KUKA KRL program: MyProgram_051().src

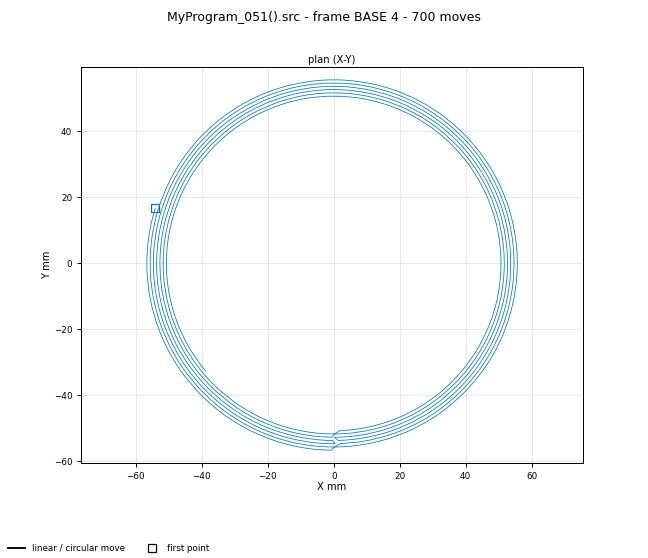
[picture p0: tool path of MyProgram_051().src in frame BASE 4, 700 of 700 moves have a stored position in this frame; points joined in program order, loops and branches not executed]
&ACCESS RVP
&REL 1
&PARAM TEMPLATE = C:\KRC\Roboter\Template\vorgabe
&PARAM EDITMASK = *
DEF MyProgram_051()
; ---- Setting reference (Base) ----
$BASE = BASE_DATA[4]

; --------------------------
; ---- Setting tool (TCP) ----
$TOOL = TOOL_DATA[3]
; --------------------------

$VEL.CP = VEL_APROX_PRINT
Startdeposition()
$VEL.CP = VEL_PRINT
LIN {X -54.1221,Y 16.7008,Z 67,A 157.6929,B 24.8675,C -2.6568,E1 24.846,E2 286.0858} C_DIS
LIN {X -55.301,Y 12.245,Z 67,A 161.7731,B 24.8699,C -2.6326,E1 24.8433,E2 282.0395} C_DIS
LIN {X -55.8838,Y 9.2265,Z 67,A 165.4414,B 24.8699,C -2.6321,E1 24.8415,E2 278.3507} C_DIS
LIN {X -56.3242,Y 5.9752,Z 67,A 168.1233,B 24.872,C -2.6111,E1 24.8406,E2 275.7029} C_DIS
LIN {X -56.6148,Y 1.6943,Z 67,A 172.8319,B 24.8727,C -2.6035,E1 24.8398,E2 270.9843} C_DIS
LIN {X -56.6219,Y -1.4652,Z 67,A 175.993,B 24.8738,C -2.5928,E1 24.8398,E2 267.8296} C_DIS
LIN {X -56.5443,Y -3.2994,Z 67,A 178.54,B 24.8732,C -2.5985,E1 24.8403,E2 265.2537} C_DIS
LIN {X -56.0863,Y -7.9019,Z 67,A -177.3263,B 24.8755,C -2.5749,E1 24.8417,E2 261.1517} C_DIS
LIN {X -55.5998,Y -10.8064,Z 67,A -174.3733,B 24.8765,C -2.5653,E1 24.8431,E2 258.2041} C_DIS
LIN {X -55.076,Y -13.2208,Z 67,A -171.0837,B 24.8759,C -2.5711,E1 24.8453,E2 254.8814} C_DIS
LIN {X -53.9542,Y -17.2366,Z 67,A -167.7374,B 24.8785,C -2.5439,E1 24.8479,E2 251.5808} C_DIS
LIN {X -53.1528,Y -19.5683,Z 67,A -165.0978,B 24.879,C -2.5391,E1 24.8504,E2 248.9377} C_DIS
LIN {X -51.9771,Y -22.5057,Z 67,A -162.0223,B 24.88,C -2.528,E1 24.8537,E2 245.8717} C_DIS
LIN {X -50.9065,Y -24.8344,Z 67,A -159.21,B 24.8804,C -2.5246,E1 24.8571,E2 243.0523} C_DIS
LIN {X -49.5347,Y -27.4672,Z 67,A -156.3958,B 24.8814,C -2.5133,E1 24.8607,E2 240.2501} C_DIS
LIN {X -48.1857,Y -29.7712,Z 67,A -153.4781,B 24.8817,C -2.5101,E1 24.865,E2 237.3252} C_DIS
LIN {X -46.639,Y -32.1398,Z 67,A -150.7212,B 24.8826,C -2.5011,E1 24.8692,E2 234.5758} C_DIS
LIN {X -45.2413,Y -34.0785,Z 67,A -147.4375,B 24.8817,C -2.5105,E1 24.8748,E2 231.2539} C_DIS
LIN {X -41.3308,Y -38.7283,Z 67,A -141.1779,B 24.8828,C -2.499,E1 24.8864,E2 224.9939} C_DIS
LIN {X -39.0762,Y -41.0032,Z 67,A -137.9651,B 24.8834,C -2.4919,E1 24.8929,E2 221.7846} C_DIS
LIN {X -35.9928,Y -43.7344,Z 67,A -134.4049,B 24.8852,C -2.4731,E1 24.9004,E2 218.2555} C_DIS
LIN {X -33.4392,Y -45.7158,Z 67,A -131.3934,B 24.8862,C -2.4628,E1 24.9071,E2 215.2577} C_DIS
LIN {X -31.3897,Y -47.1472,Z 67,A -128.7043,B 24.8862,C -2.4618,E1 24.9133,E2 212.5622} C_DIS
LIN {X -29.065,Y -48.615,Z 67,A -125.9136,B 24.8866,C -2.4579,E1 24.92,E2 209.772} C_DIS
LIN {X -26.584,Y -50.0145,Z 67,A -123.2284,B 24.8873,C -2.4505,E1 24.9265,E2 207.0968} C_DIS
LIN {X -24.2627,Y -51.1812,Z 67,A -120.5751,B 24.8875,C -2.4478,E1 24.9332,E2 204.4429} C_DIS
LIN {X -20.1408,Y -52.9383,Z 67,A -115.6937,B 24.8874,C -2.4499,E1 24.9458,E2 199.5456} C_DIS
LIN {X -16.9667,Y -54.0396,Z 67,A -112.4919,B 24.8879,C -2.4435,E1 24.9543,E2 196.3531} C_DIS
LIN {X -14.3599,Y -54.7903,Z 67,A -109.8261,B 24.8882,C -2.4403,E1 24.9615,E2 193.6907} C_DIS
LIN {X -11.9749,Y -55.3599,Z 67,A -107.3588,B 24.8884,C -2.4389,E1 24.9682,E2 191.2237} C_DIS
LIN {X -9.3697,Y -55.8598,Z 67,A -104.6044,B 24.8884,C -2.4394,E1 24.9758,E2 188.4653} C_DIS
LIN {X -6.5203,Y -56.2637,Z 67,A -101.862,B 24.8887,C -2.4355,E1 24.9833,E2 185.73} C_DIS
LIN {X -4.0645,Y -56.4947,Z 67,A -99.183,B 24.8883,C -2.4391,E1 24.9908,E2 183.0414} C_DIS
LIN {X -0.895,Y -56.6333,Z 67,A -95.9984,B 24.8883,C -2.4391,E1 24.9997,E2 179.8564} C_DIS
LIN {X -0.895,Y -56.6333,Z 67,A -95.9984,B 24.8883,C -2.4391,E1 24.9997,E2 179.8564} C_DIS
Enddeposition()
LIN {X 0.3106,Y -55.6512,Z 67,A -94.8837,B 24.887,C -2.4541,E1 25.0029,E2 178.706} C_DIS
Startdeposition()
$VEL.CP = VEL_PRINT
LIN {X -1.8445,Y -55.6223,Z 67,A -98.806,B 24.89,C -2.4206,E1 24.9918,E2 182.7081} C_DIS
LIN {X -4.7912,Y -55.447,Z 67,A -101.3708,B 24.8892,C -2.4297,E1 24.9847,E2 185.2525} C_DIS
LIN {X -7.4963,Y -55.1465,Z 67,A -104.2719,B 24.8893,C -2.4282,E1 24.9766,E2 188.159} C_DIS
LIN {X -11.1478,Y -54.5248,Z 67,A -108.48,B 24.8899,C -2.4223,E1 24.965,E2 192.3859} C_DIS
LIN {X -13.8894,Y -53.8916,Z 67,A -110.9193,B 24.889,C -2.4323,E1 24.9585,E2 194.8048} C_DIS
LIN {X -16.4128,Y -53.1775,Z 67,A -113.7184,B 24.889,C -2.4323,E1 24.9509,E2 197.6086} C_DIS
LIN {X -18.8336,Y -52.3696,Z 67,A -116.0432,B 24.8883,C -2.4399,E1 24.9448,E2 199.9195} C_DIS
LIN {X -21.0409,Y -51.5219,Z 67,A -118.81,B 24.8886,C -2.4362,E1 24.9376,E2 202.7012} C_DIS
LIN {X -23.8797,Y -50.2697,Z 67,A -121.8951,B 24.8881,C -2.4417,E1 24.9298,E2 205.7808} C_DIS
LIN {X -26.7603,Y -48.7973,Z 67,A -124.7977,B 24.887,C -2.4535,E1 24.9227,E2 208.6632} C_DIS
LIN {X -29.3984,Y -47.2542,Z 67,A -128.3435,B 24.8873,C -2.4509,E1 24.9141,E2 212.226} C_DIS
LIN {X -31.6691,Y -45.7635,Z 67,A -131.1634,B 24.8869,C -2.4549,E1 24.9076,E2 215.0458} C_DIS
LIN {X -34.5559,Y -43.6247,Z 67,A -134.6556,B 24.886,C -2.4649,E1 24.8998,E2 218.5269} C_DIS
LIN {X -36.5148,Y -41.9989,Z 67,A -138.1181,B 24.8868,C -2.4554,E1 24.8924,E2 222.0254} C_DIS
LIN {X -40.0607,Y -38.6311,Z 67,A -142.3125,B 24.8846,C -2.4799,E1 24.8841,E2 226.1788} C_DIS
LIN {X -41.1545,Y -37.4636,Z 67,A -144.6872,B 24.8854,C -2.4713,E1 24.8796,E2 228.5847} C_DIS
LIN {X -44.1926,Y -33.827,Z 67,A -149.3108,B 24.8839,C -2.4868,E1 24.8715,E2 233.1927} C_DIS
LIN {X -45.5071,Y -32.038,Z 67,A -151.4004,B 24.8831,C -2.4956,E1 24.8681,E2 235.2717} C_DIS
LIN {X -47.4442,Y -29.0915,Z 67,A -154.6624,B 24.8817,C -2.5108,E1 24.8632,E2 238.5137} C_DIS
LIN {X -48.5041,Y -27.2875,Z 67,A -157.3262,B 24.8819,C -2.5081,E1 24.8595,E2 241.1977} C_DIS
LIN {X -49.835,Y -24.7729,Z 67,A -160.2896,B 24.8812,C -2.5155,E1 24.8557,E2 244.1595} C_DIS
LIN {X -51.5972,Y -20.856,Z 67,A -164.7992,B 24.8802,C -2.5265,E1 24.8507,E2 248.6677} C_DIS
LIN {X -52.3478,Y -18.8934,Z 67,A -166.8741,B 24.8795,C -2.5341,E1 24.8487,E2 250.7361} C_DIS
LIN {X -53.23,Y -16.2436,Z 67,A -170.2299,B 24.8794,C -2.5349,E1 24.8459,E2 254.1092} C_DIS
LIN {X -54.2859,Y -12.2611,Z 67,A -173.8372,B 24.8772,C -2.5577,E1 24.8434,E2 257.6831} C_DIS
LIN {X -54.8971,Y -9.137,Z 67,A -177.5377,B 24.8769,C -2.561,E1 24.8416,E2 261.3975} C_DIS
LIN {X -55.3786,Y -5.5122,Z 67,A 178.4718,B 24.8761,C -2.5692,E1 24.8403,E2 265.3924} C_DIS
LIN {X -55.6028,Y -2.3569,Z 67,A 175.2683,B 24.875,C -2.5802,E1 24.8398,E2 268.5889} C_DIS
LIN {X -55.6332,Y 1.4878,Z 67,A 171.6315,B 24.8733,C -2.5977,E1 24.8398,E2 272.2058} C_DIS
LIN {X -55.4904,Y 4.2453,Z 67,A 169.0616,B 24.872,C -2.6109,E1 24.8403,E2 274.7594} C_DIS
LIN {X -55.353,Y 5.7673,Z 67,A 167.1882,B 24.872,C -2.6112,E1 24.8408,E2 276.6435} C_DIS
LIN {X -55.0287,Y 8.313,Z 67,A 164.6327,B 24.871,C -2.6208,E1 24.8418,E2 279.1912} C_DIS
LIN {X -54.6417,Y 10.5596,Z 67,A 161.8621,B 24.871,C -2.6216,E1 24.8432,E2 281.9764} C_DIS
LIN {X -53.7999,Y 14.2433,Z 67,A 157.9782,B 24.8698,C -2.6337,E1 24.8458,E2 285.854} C_DIS
LIN {X -53.2007,Y 16.3381,Z 67,A 155.4974,B 24.8694,C -2.6369,E1 24.8479,E2 288.3415} C_DIS
LIN {X -52.3409,Y 18.9123,Z 67,A 152.2747,B 24.8693,C -2.6387,E1 24.8509,E2 291.5781} C_DIS
LIN {X -50.5816,Y 23.2124,Z 67,A 148.3561,B 24.8665,C -2.6664,E1 24.8552,E2 295.4521} C_DIS
LIN {X -49.413,Y 25.6061,Z 67,A 145.5521,B 24.8658,C -2.6734,E1 24.8587,E2 298.2545} C_DIS
LIN {X -48.1498,Y 27.9081,Z 67,A 142.8105,B 24.8651,C -2.6805,E1 24.8625,E2 300.9935} C_DIS
LIN {X -46.6638,Y 30.3274,Z 67,A 139.9688,B 24.8641,C -2.6899,E1 24.8667,E2 303.8273} C_DIS
LIN {X -44.8507,Y 32.9491,Z 67,A 136.9036,B 24.8629,C -2.7022,E1 24.8716,E2 306.8781} C_DIS
LIN {X -43.6109,Y 34.5734,Z 67,A 134.4878,B 24.8629,C -2.7026,E1 24.8758,E2 309.3042} C_DIS
LIN {X -41.8572,Y 36.677,Z 67,A 131.7034,B 24.862,C -2.7103,E1 24.8808,E2 312.083} C_DIS
LIN {X -39.6827,Y 39.0195,Z 67,A 128.1736,B 24.8616,C -2.7143,E1 24.8876,E2 315.6185} C_DIS
LIN {X -37.3353,Y 41.272,Z 67,A 124.9518,B 24.8606,C -2.7241,E1 24.8942,E2 318.8301} C_DIS
LIN {X -35.221,Y 43.0901,Z 67,A 122.1383,B 24.8599,C -2.7313,E1 24.9002,E2 321.6372} C_DIS
LIN {X -33.067,Y 44.7644,Z 67,A 119.0584,B 24.8598,C -2.7325,E1 24.9071,E2 324.7253} C_DIS
LIN {X -29.6626,Y 47.0892,Z 67,A 115.4695,B 24.8578,C -2.7517,E1 24.9153,E2 328.2803} C_DIS
LIN {X -26.8663,Y 48.7393,Z 67,A 111.6008,B 24.8581,C -2.7485,E1 24.9247,E2 332.1681} C_DIS
LIN {X -24.4566,Y 49.9918,Z 67,A 108.8439,B 24.8576,C -2.7536,E1 24.9316,E2 334.9201} C_DIS
LIN {X -21.7856,Y 51.2118,Z 67,A 105.258,B 24.8581,C -2.7483,E1 24.9408,E2 338.5272} C_DIS
LIN {X -18.7901,Y 52.3853,Z 67,A 102.8014,B 24.8561,C -2.7675,E1 24.9471,E2 340.9433} C_DIS
LIN {X -15.8274,Y 53.3546,Z 67,A 98.6582,B 24.8575,C -2.7546,E1 24.9583,E2 345.1243} C_DIS
LIN {X -12.7972,Y 54.1618,Z 67,A 95.4033,B 24.8572,C -2.7571,E1 24.9671,E2 348.3777} C_DIS
LIN {X -7.566,Y 55.1364,Z 67,A 90.5156,B 24.8557,C -2.7717,E1 24.9805,E2 353.2354} C_DIS
LIN {X -4.5272,Y 55.4683,Z 67,A 87.2828,B 24.8557,C -2.7717,E1 24.9894,E2 356.4699} C_DIS
LIN {X -1.7783,Y 55.6243,Z 67,A 84.466,B 24.8556,C -2.7729,E1 24.9973,E2 359.2843} C_DIS
LIN {X 1.3657,Y 55.637,Z 67,A 81.6491,B 24.8547,C -2.7813,E1 25.0051,E2 362.0811} C_DIS
LIN {X 3.1678,Y 55.5625,Z 67,A 79.4313,B 24.8554,C -2.7746,E1 25.0113,E2 364.3141} C_DIS
LIN {X 5.966,Y 55.3322,Z 67,A 76.2287,B 24.856,C -2.7684,E1 25.0203,E2 367.5295} C_DIS
LIN {X 10.5629,Y 54.6411,Z 67,A 71.7775,B 24.8555,C -2.7733,E1 25.0325,E2 371.9646} C_DIS
LIN {X 13.0854,Y 54.0926,Z 67,A 68.9473,B 24.856,C -2.7685,E1 25.0402,E2 374.8021} C_DIS
LIN {X 15.7507,Y 53.3774,Z 67,A 66.5106,B 24.8554,C -2.7746,E1 25.0467,E2 377.2205} C_DIS
LIN {X 18.0833,Y 52.6324,Z 67,A 63.5248,B 24.8566,C -2.7634,E1 25.0547,E2 380.2271} C_DIS
LIN {X 20.7445,Y 51.6425,Z 67,A 60.8487,B 24.8564,C -2.7655,E1 25.0616,E2 382.8924} C_DIS
LIN {X 23.7433,Y 50.3345,Z 67,A 57.4715,B 24.8568,C -2.7615,E1 25.0702,E2 386.2705} C_DIS
LIN {X 26.1701,Y 49.1164,Z 67,A 54.7715,B 24.8569,C -2.7599,E1 25.0769,E2 388.9668} C_DIS
LIN {X 28.4356,Y 47.8399,Z 67,A 52.0436,B 24.8574,C -2.7551,E1 25.0835,E2 391.6979} C_DIS
LIN {X 30.7794,Y 46.3668,Z 67,A 49.258,B 24.8577,C -2.752,E1 25.09,E2 394.4817} C_DIS
LIN {X 32.7053,Y 45.0292,Z 67,A 46.9243,B 24.858,C -2.7497,E1 25.0953,E2 396.8128} C_DIS
LIN {X 35.9425,Y 42.4899,Z 67,A 42.7233,B 24.8587,C -2.7427,E1 25.1045,E2 401.0146} C_DIS
LIN {X 38.4218,Y 40.2624,Z 67,A 39.2402,B 24.8595,C -2.7349,E1 25.1117,E2 404.5023} C_DIS
LIN {X 40.6729,Y 37.9865,Z 67,A 36.2169,B 24.8596,C -2.7336,E1 25.1176,E2 407.5155} C_DIS
LIN {X 43.1485,Y 35.149,Z 67,A 32.5217,B 24.8601,C -2.7288,E1 25.1243,E2 411.2054} C_DIS
LIN {X 44.2479,Y 33.754,Z 67,A 29.9013,B 24.8623,C -2.7075,E1 25.1288,E2 413.8638} C_DIS
LIN {X 46.5073,Y 30.5663,Z 67,A 26.43,B 24.8621,C -2.7094,E1 25.1343,E2 417.3136} C_DIS
LIN {X 47.6256,Y 28.7931,Z 67,A 24.4975,B 24.8622,C -2.7088,E1 25.1371,E2 419.2378} C_DIS
LIN {X 48.5299,Y 27.2412,Z 67,A 22.2207,B 24.8636,C -2.6946,E1 25.1403,E2 421.5363} C_DIS
LIN {X 49.765,Y 24.9142,Z 67,A 19.2963,B 24.8649,C -2.6826,E1 25.1441,E2 424.4735} C_DIS
LIN {X 50.9938,Y 22.2902,Z 67,A 16.8273,B 24.8646,C -2.6856,E1 25.1469,E2 426.9222} C_DIS
LIN {X 52.4735,Y 18.541,Z 67,A 12.9781,B 24.8651,C -2.6803,E1 25.1508,E2 430.7625} C_DIS
LIN {X 53.1743,Y 16.4231,Z 67,A 9.8911,B 24.8675,C -2.6561,E1 25.1535,E2 433.8891} C_DIS
LIN {X 53.8261,Y 14.1443,Z 67,A 7.7022,B 24.8677,C -2.6544,E1 25.155,E2 436.0696} C_DIS
LIN {X 54.454,Y 11.4927,Z 67,A 4.92,B 24.8685,C -2.6464,E1 25.1567,E2 438.8546} C_DIS
LIN {X 55.0641,Y 8.0767,Z 67,A 1.1075,B 24.8701,C -2.6301,E1 25.1585,E2 442.6832} C_DIS
LIN {X 55.4353,Y 4.9183,Z 67,A -1.8284,B 24.8704,C -2.6274,E1 25.1593,E2 445.6081} C_DIS
LIN {X 55.5989,Y 2.4463,Z 67,A -4.3077,B 24.871,C -2.621,E1 25.1597,E2 448.0878} C_DIS
LIN {X 55.6492,Y -0.7025,Z 67,A -7.5822,B 24.8721,C -2.61,E1 25.1597,E2 451.3687} C_DIS
LIN {X 55.5487,Y -3.4141,Z 67,A -10.1765,B 24.8725,C -2.6057,E1 25.1594,E2 453.9579} C_DIS
LIN {X 55.3691,Y -5.6137,Z 67,A -12.6549,B 24.8737,C -2.5939,E1 25.1588,E2 456.4495} C_DIS
LIN {X 54.6207,Y -10.6686,Z 67,A -17.6644,B 24.8747,C -2.583,E1 25.1566,E2 461.4554} C_DIS
LIN {X 53.8338,Y -14.1146,Z 67,A -21.8632,B 24.877,C -2.5592,E1 25.1538,E2 465.6861} C_DIS
LIN {X 52.8671,Y -17.3885,Z 67,A -24.9749,B 24.8772,C -2.5573,E1 25.1512,E2 468.7845} C_DIS
LIN {X 51.5397,Y -20.9972,Z 67,A -28.8243,B 24.8781,C -2.5478,E1 25.1474,E2 472.6351} C_DIS
LIN {X 50.5576,Y -23.2629,Z 67,A -31.647,B 24.8795,C -2.534,E1 25.1441,E2 475.4749} C_DIS
LIN {X 49.3194,Y -25.7846,Z 67,A -34.155,B 24.8795,C -2.534,E1 25.141,E2 477.9695} C_DIS
LIN {X 48.0794,Y -28.0304,Z 67,A -37.0219,B 24.8806,C -2.5216,E1 25.137,E2 480.8511} C_DIS
LIN {X 46.3184,Y -30.8518,Z 67,A -40.2414,B 24.8811,C -2.5166,E1 25.1322,E2 484.0662} C_DIS
LIN {X 45.1277,Y -32.569,Z 67,A -42.7948,B 24.8825,C -2.502,E1 25.128,E2 486.6417} C_DIS
LIN {X 42.5488,Y -35.8734,Z 67,A -46.3701,B 24.882,C -2.5069,E1 25.1218,E2 490.1887} C_DIS
LIN {X 40.8122,Y -37.8374,Z 67,A -49.8027,B 24.8842,C -2.4843,E1 25.1153,E2 493.6596} C_DIS
LIN {X 38.8834,Y -39.8163,Z 67,A -52.617,B 24.8847,C -2.4782,E1 25.1097,E2 496.4765} C_DIS
LIN {X 35.7352,Y -42.6646,Z 67,A -56.1642,B 24.884,C -2.4859,E1 25.1024,E2 499.9911} C_DIS
LIN {X 33.6953,Y -44.2937,Z 67,A -59.657,B 24.8861,C -2.4631,E1 25.0946,E2 503.5252} C_DIS
LIN {X 31.2855,Y -46.0266,Z 67,A -62.2486,B 24.8858,C -2.4668,E1 25.0887,E2 506.0991} C_DIS
LIN {X 29.2788,Y -47.329,Z 67,A -64.7057,B 24.8862,C -2.4623,E1 25.0829,E2 508.5589} C_DIS
LIN {X 27.4558,Y -48.4097,Z 67,A -66.8391,B 24.8865,C -2.4594,E1 25.0777,E2 510.6926} C_DIS
LIN {X 24.5983,Y -49.9216,Z 67,A -70.2743,B 24.8872,C -2.4517,E1 25.0692,E2 514.1366} C_DIS
LIN {X 22.1325,Y -51.0626,Z 67,A -73.1308,B 24.8877,C -2.4463,E1 25.0619,E2 516.9988} C_DIS
LIN {X 19.0744,Y -52.2818,Z 67,A -76.7513,B 24.8885,C -2.4371,E1 25.0524,E2 520.6335} C_DIS
LIN {X 16.1825,Y -53.2489,Z 67,A -79.5818,B 24.8883,C -2.4396,E1 25.0449,E2 523.4526} C_DIS
LIN {X 11.9676,Y -54.3508,Z 67,A -84.3187,B 24.8892,C -2.4302,E1 25.032,E2 528.2049} C_DIS
LIN {X 9.1373,Y -54.8975,Z 67,A -87.3514,B 24.8895,C -2.4267,E1 25.0237,E2 531.2429} C_DIS
LIN {X 5.1568,Y -55.4133,Z 67,A -90.8379,B 24.8885,C -2.4369,E1 25.0141,E2 534.7024} C_DIS
LIN {X 2.997,Y -55.572,Z 67,A -93.4015,B 24.8892,C -2.4294,E1 25.0069,E2 537.2828} C_DIS
LIN {X 0.3106,Y -55.6512,Z 67,A -94.883,B 24.887,C -2.4538,E1 25.0029,E2 538.706} C_DIS
Enddeposition()
LIN {X 0.3106,Y -55.6512,Z 67,A -94.883,B 24.887,C -2.4538,E1 25.0029,E2 538.706} C_DIS
Startdeposition()
$VEL.CP = VEL_PRINT
LIN {X 1.9823,Y -54.63,Z 67,A -92.5802,B 24.8844,C -2.4821,E1 25.0095,E2 536.3366} C_DIS
LIN {X 7.2815,Y -54.1787,Z 67,A -86.6921,B 24.8835,C -2.4915,E1 25.0259,E2 530.4302} C_DIS
LIN {X 11.5086,Y -53.4402,Z 67,A -82.6061,B 24.8839,C -2.487,E1 25.0371,E2 526.3599} C_DIS
LIN {X 15.7752,Y -52.34,Z 67,A -78.3873,B 24.8842,C -2.4837,E1 25.0484,E2 522.1557} C_DIS
LIN {X 18.8016,Y -51.3302,Z 67,A -74.9215,B 24.8836,C -2.4904,E1 25.0575,E2 518.681} C_DIS
LIN {X 21.2357,Y -50.3719,Z 67,A -72.2364,B 24.8833,C -2.4931,E1 25.0645,E2 515.9957} C_DIS
LIN {X 23.9977,Y -49.1171,Z 67,A -69.529,B 24.8838,C -2.4882,E1 25.0713,E2 513.3069} C_DIS
LIN {X 25.9093,Y -48.1355,Z 67,A -66.7457,B 24.8824,C -2.503,E1 25.0782,E2 510.4962} C_DIS
LIN {X 28.0377,Y -46.928,Z 67,A -64.5615,B 24.8827,C -2.4996,E1 25.0834,E2 508.3267} C_DIS
LIN {X 30.5521,Y -45.3306,Z 67,A -61.5262,B 24.8823,C -2.5037,E1 25.0906,E2 505.2917} C_DIS
LIN {X 31.8249,Y -44.4463,Z 67,A -59.4378,B 24.8811,C -2.5169,E1 25.0954,E2 503.1795} C_DIS
LIN {X 34.6629,Y -42.2713,Z 67,A -55.9867,B 24.8809,C -2.5185,E1 25.1029,E2 499.7373} C_DIS
LIN {X 36.6555,Y -40.5549,Z 67,A -53.1679,B 24.8802,C -2.526,E1 25.1088,E2 496.9118} C_DIS
LIN {X 38.4223,Y -38.8845,Z 67,A -50.8245,B 24.8801,C -2.5276,E1 25.1135,E2 494.5744} C_DIS
LIN {X 40.1119,Y -37.1398,Z 67,A -48.0166,B 24.8789,C -2.5395,E1 25.1189,E2 491.7506} C_DIS
LIN {X 41.8499,Y -35.1705,Z 67,A -45.1235,B 24.878,C -2.5496,E1 25.1242,E2 488.8468} C_DIS
LIN {X 44.048,Y -32.3739,Z 67,A -41.951,B 24.8782,C -2.5472,E1 25.1296,E2 485.6949} C_DIS
LIN {X 44.9481,Y -31.1121,Z 67,A -39.6945,B 24.8764,C -2.5655,E1 25.1332,E2 483.4062} C_DIS
LIN {X 46.4624,Y -28.8021,Z 67,A -37.0281,B 24.8761,C -2.5685,E1 25.1372,E2 480.7461} C_DIS
LIN {X 48.002,Y -26.1553,Z 67,A -33.9945,B 24.8756,C -2.5738,E1 25.1413,E2 477.7158} C_DIS
LIN {X 49.9347,Y -22.2444,Z 67,A -29.7776,B 24.8751,C -2.5794,E1 25.1464,E2 473.5085} C_DIS
LIN {X 50.5459,Y -20.8195,Z 67,A -27.6895,B 24.8736,C -2.5945,E1 25.1487,E2 471.396} C_DIS
LIN {X 51.7095,Y -17.7312,Z 67,A -24.4821,B 24.8731,C -2.5994,E1 25.1517,E2 468.195} C_DIS
LIN {X 52.63,Y -14.7776,Z 67,A -20.9799,B 24.8716,C -2.6152,E1 25.1545,E2 464.6754} C_DIS
LIN {X 53.2679,Y -12.2805,Z 67,A -18.498,B 24.8712,C -2.6187,E1 25.1561,E2 462.1997} C_DIS
LIN {X 54.0301,Y -8.3088,Z 67,A -13.4497,B 24.8681,C -2.6502,E1 25.1585,E2 457.1065} C_DIS
LIN {X 54.4502,Y -4.8468,Z 67,A -10.1854,B 24.8678,C -2.6529,E1 25.1594,E2 453.8552} C_DIS
LIN {X 54.6616,Y -0.7001,Z 67,A -6.335,B 24.8676,C -2.6554,E1 25.1598,E2 450.0218} C_DIS
LIN {X 54.6069,Y 2.5302,Z 67,A -2.9419,B 24.8665,C -2.6662,E1 25.1595,E2 446.6234} C_DIS
LIN {X 54.4176,Y 5.2003,Z 67,A -0.0277,B 24.8654,C -2.6773,E1 25.1588,E2 443.7} C_DIS
LIN {X 54.0544,Y 8.1511,Z 67,A 2.991,B 24.8646,C -2.6848,E1 25.1577,E2 440.6815} C_DIS
LIN {X 53.451,Y 11.4591,Z 67,A 6.4254,B 24.8638,C -2.6935,E1 25.1558,E2 437.2464} C_DIS
LIN {X 52.8997,Y 13.7819,Z 67,A 9.332,B 24.8621,C -2.71,E1 25.1538,E2 434.3176} C_DIS
LIN {X 51.7356,Y 17.6565,Z 67,A 12.7943,B 24.8626,C -2.7053,E1 25.1509,E2 430.8861} C_DIS
LIN {X 50.523,Y 20.8755,Z 67,A 16.3678,B 24.8616,C -2.7149,E1 25.1473,E2 427.3097} C_DIS
LIN {X 49.6029,Y 22.9749,Z 67,A 19.7066,B 24.8588,C -2.7421,E1 25.1434,E2 423.9246} C_DIS
LIN {X 47.8274,Y 26.4739,Z 67,A 23.1375,B 24.8592,C -2.7383,E1 25.1389,E2 420.521} C_DIS
LIN {X 46.9068,Y 28.0736,Z 67,A 25.2669,B 24.8582,C -2.7475,E1 25.1359,E2 418.3806} C_DIS
LIN {X 45.2055,Y 30.7369,Z 67,A 28.3637,B 24.8578,C -2.7512,E1 25.1312,E2 415.2906} C_DIS
LIN {X 43.6371,Y 32.9256,Z 67,A 31.2361,B 24.857,C -2.7591,E1 25.1264,E2 412.4133} C_DIS
LIN {X 42.0608,Y 34.9166,Z 67,A 33.8427,B 24.8565,C -2.7641,E1 25.1218,E2 409.807} C_DIS
LIN {X 40.4202,Y 36.8039,Z 67,A 36.5279,B 24.8557,C -2.7712,E1 25.1168,E2 407.1168} C_DIS
LIN {X 38.2385,Y 39.0661,Z 67,A 39.5381,B 24.8557,C -2.7722,E1 25.1109,E2 404.1172} C_DIS
LIN {X 36.3351,Y 40.8417,Z 67,A 42.4814,B 24.8546,C -2.7821,E1 25.1048,E2 401.1623} C_DIS
LIN {X 34.3582,Y 42.5183,Z 67,A 45.1302,B 24.8542,C -2.7857,E1 25.0991,E2 398.5151} C_DIS
LIN {X 32.3895,Y 44.0365,Z 67,A 47.5643,B 24.8542,C -2.7866,E1 25.0937,E2 396.0875} C_DIS
LIN {X 29.4791,Y 46.0355,Z 67,A 51.5502,B 24.8529,C -2.7984,E1 25.0844,E2 392.0872} C_DIS
LIN {X 26.8906,Y 47.5947,Z 67,A 54.6311,B 24.8526,C -2.8011,E1 25.077,E2 389.0092} C_DIS
LIN {X 24.5763,Y 48.8303,Z 67,A 57.0754,B 24.8529,C -2.7984,E1 25.071,E2 386.578} C_DIS
LIN {X 21.5913,Y 50.2213,Z 67,A 61.075,B 24.8513,C -2.8133,E1 25.0607,E2 382.5531} C_DIS
LIN {X 19.1158,Y 51.2146,Z 67,A 63.6987,B 24.8514,C -2.8124,E1 25.0539,E2 379.9371} C_DIS
LIN {X 16.4547,Y 52.1306,Z 67,A 66.939,B 24.8506,C -2.8205,E1 25.0453,E2 376.6837} C_DIS
LIN {X 12.0362,Y 53.3243,Z 67,A 71.2728,B 24.8512,C -2.8142,E1 25.0336,E2 372.3714} C_DIS
LIN {X 8.8669,Y 53.9415,Z 67,A 74.9893,B 24.8504,C -2.8219,E1 25.0233,E2 368.6407} C_DIS
LIN {X 6.2275,Y 54.3095,Z 67,A 78.5894,B 24.8487,C -2.8379,E1 25.0133,E2 365.0051} C_DIS
LIN {X 2.6694,Y 54.6009,Z 67,A 81.0955,B 24.8512,C -2.8143,E1 25.0064,E2 362.5561} C_DIS
LIN {X -1.0424,Y 54.6552,Z 67,A 84.8338,B 24.8516,C -2.8108,E1 24.996,E2 358.8265} C_DIS
LIN {X -2.6547,Y 54.6016,Z 67,A 86.9733,B 24.8508,C -2.8185,E1 24.99,E2 356.6681} C_DIS
LIN {X -5.9581,Y 54.3393,Z 67,A 90.1154,B 24.8516,C -2.8108,E1 24.9813,E2 353.5429} C_DIS
LIN {X -7.9298,Y 54.0872,Z 67,A 92.114,B 24.8519,C -2.8079,E1 24.9758,E2 351.5495} C_DIS
LIN {X -10.3945,Y 53.6679,Z 67,A 95.1561,B 24.8513,C -2.8136,E1 24.9674,E2 348.4907} C_DIS
LIN {X -12.7914,Y 53.1478,Z 67,A 97.2945,B 24.8524,C -2.8035,E1 24.9616,E2 346.3735} C_DIS
LIN {X -15.5324,Y 52.4121,Z 67,A 100.8773,B 24.8515,C -2.8113,E1 24.9519,E2 342.7665} C_DIS
LIN {X -18.5545,Y 51.4203,Z 67,A 103.8709,B 24.8526,C -2.8012,E1 24.9441,E2 339.7912} C_DIS
LIN {X -21.0677,Y 50.4427,Z 67,A 106.8461,B 24.8527,C -2.8,E1 24.9364,E2 336.8123} C_DIS
LIN {X -23.8238,Y 49.201,Z 67,A 109.98,B 24.8533,C -2.7946,E1 24.9285,E2 333.6834} C_DIS
LIN {X -26.3414,Y 47.9011,Z 67,A 112.8954,B 24.8539,C -2.7887,E1 24.9213,E2 330.7739} C_DIS
LIN {X -28.1411,Y 46.8663,Z 67,A 115.472,B 24.8536,C -2.7917,E1 24.9151,E2 328.1822} C_DIS
LIN {X -31.1429,Y 44.9267,Z 67,A 118.7379,B 24.8552,C -2.7764,E1 24.9076,E2 324.942} C_DIS
LIN {X -33.2316,Y 43.4047,Z 67,A 121.5719,B 24.8556,C -2.773,E1 24.9012,E2 322.106} C_DIS
LIN {X -35.3519,Y 41.6959,Z 67,A 124.4553,B 24.8562,C -2.7674,E1 24.895,E2 319.2252} C_DIS
LIN {X -37.2321,Y 40.0267,Z 67,A 127.7188,B 24.8557,C -2.7718,E1 24.8883,E2 315.9378} C_DIS
LIN {X -40.9282,Y 36.2389,Z 67,A 132.6533,B 24.8581,C -2.7482,E1 24.8789,E2 311.0382} C_DIS
LIN {X -42.6144,Y 34.2396,Z 67,A 135.4081,B 24.8588,C -2.7414,E1 24.874,E2 308.2868} C_DIS
LIN {X -43.7615,Y 32.76,Z 67,A 137.5181,B 24.8591,C -2.7387,E1 24.8705,E2 306.1733} C_DIS
LIN {X -45.47,Y 30.3447,Z 67,A 140.255,B 24.8606,C -2.7244,E1 24.8661,E2 303.4569} C_DIS
LIN {X -46.3436,Y 28.9923,Z 67,A 142.3432,B 24.8604,C -2.7262,E1 24.863,E2 301.3538} C_DIS
LIN {X -48.2524,Y 25.6914,Z 67,A 146.2615,B 24.8617,C -2.7136,E1 24.8577,E2 297.4452} C_DIS
LIN {X -49.8166,Y 22.5077,Z 67,A 150.1592,B 24.8625,C -2.7056,E1 24.853,E2 293.5454} C_DIS
LIN {X -50.8394,Y 20.0902,Z 67,A 152.8049,B 24.8635,C -2.6957,E1 24.8503,E2 290.9087} C_DIS
LIN {X -52.4082,Y 15.5455,Z 67,A 157.948,B 24.8649,C -2.6819,E1 24.8458,E2 285.7691} C_DIS
LIN {X -53.1864,Y 12.6333,Z 67,A 161.8085,B 24.8648,C -2.6833,E1 24.8432,E2 281.8828} C_DIS
LIN {X -53.8355,Y 9.4901,Z 67,A 164.8061,B 24.8664,C -2.6669,E1 24.8417,E2 278.9066} C_DIS
LIN {X -54.3819,Y 5.5595,Z 67,A 168.4825,B 24.8685,C -2.6461,E1 24.8404,E2 275.2578} C_DIS
LIN {X -54.5701,Y 3.2166,Z 67,A 170.8645,B 24.8694,C -2.6371,E1 24.84,E2 272.8831} C_DIS
LIN {X -54.6509,Y 1.2776,Z 67,A 173.0569,B 24.8698,C -2.6332,E1 24.8398,E2 270.6869} C_DIS
LIN {X -54.6475,Y -1.4145,Z 67,A 176.144,B 24.8703,C -2.6285,E1 24.8399,E2 267.5924} C_DIS
LIN {X -54.4784,Y -4.5092,Z 67,A 179.3286,B 24.8714,C -2.6174,E1 24.8405,E2 264.4153} C_DIS
LIN {X -54.1418,Y -7.5475,Z 67,A -177.4963,B 24.8724,C -2.607,E1 24.8416,E2 261.246} C_DIS
LIN {X -53.6425,Y -10.5264,Z 67,A -174.5405,B 24.8737,C -2.594,E1 24.8431,E2 258.3038} C_DIS
LIN {X -53.0306,Y -13.2656,Z 67,A -171.4096,B 24.8742,C -2.5881,E1 24.8451,E2 255.1685} C_DIS
LIN {X -52.1921,Y -16.2566,Z 67,A -168.1325,B 24.8751,C -2.5788,E1 24.8477,E2 251.8948} C_DIS
LIN {X -51.4239,Y -18.5448,Z 67,A -165.485,B 24.8757,C -2.5734,E1 24.8501,E2 249.2453} C_DIS
LIN {X -50.5403,Y -20.8328,Z 67,A -162.6153,B 24.8759,C -2.5709,E1 24.8531,E2 246.3654} C_DIS
LIN {X -48.5848,Y -25.0568,Z 67,A -158.1155,B 24.8778,C -2.5513,E1 24.8586,E2 241.8879} C_DIS
LIN {X -46.6738,Y -28.4578,Z 67,A -154.2195,B 24.8791,C -2.5375,E1 24.864,E2 238.0048} C_DIS
LIN {X -45.6755,Y -30.034,Z 67,A -151.8455,B 24.8789,C -2.5394,E1 24.8676,E2 235.6141} C_DIS
LIN {X -44.4694,Y -31.7924,Z 67,A -149.3054,B 24.8789,C -2.5391,E1 24.8717,E2 233.0625} C_DIS
LIN {X -42.0307,Y -34.9529,Z 67,A -145.3826,B 24.8803,C -2.525,E1 24.8785,E2 229.155} C_DIS
LIN {X -40.4663,Y -36.7534,Z 67,A -143.2395,B 24.8814,C -2.5134,E1 24.8825,E2 227.0298} C_DIS
LIN {X -39.3468,Y -37.9488,Z 67,A -141.6009,B 24.8819,C -2.5085,E1 24.8856,E2 225.3959} C_DIS
LIN {X -37.6038,Y -39.6772,Z 67,A -138.3358,B 24.8813,C -2.5151,E1 24.8922,E2 222.1015} C_DIS
LIN {X -34.5911,Y -42.3295,Z 67,A -134.4223,B 24.8825,C -2.5021,E1 24.9005,E2 218.2038} C_DIS
LIN {X -31.7218,Y -44.5198,Z 67,A -130.6227,B 24.8831,C -2.496,E1 24.909,E2 214.4053} C_DIS
LIN {X -29.2783,Y -46.1644,Z 67,A -127.5602,B 24.8836,C -2.4908,E1 24.9162,E2 211.3452} C_DIS
LIN {X -27.1162,Y -47.4659,Z 67,A -124.8403,B 24.8838,C -2.4884,E1 24.9228,E2 208.6227} C_DIS
LIN {X -24.621,Y -48.8075,Z 67,A -121.6663,B 24.8838,C -2.4884,E1 24.9307,E2 205.4402} C_DIS
LIN {X -21.8407,Y -50.1125,Z 67,A -118.6326,B 24.8844,C -2.4816,E1 24.9384,E2 202.4154} C_DIS
LIN {X -19.4462,Y -51.0895,Z 67,A -115.723,B 24.8844,C -2.4827,E1 24.946,E2 199.4969} C_DIS
LIN {X -15.5881,Y -52.3956,Z 67,A -111.676,B 24.885,C -2.4754,E1 24.9567,E2 195.4601} C_DIS
LIN {X -13.728,Y -52.9135,Z 67,A -109.4222,B 24.8847,C -2.4785,E1 24.9628,E2 193.1955} C_DIS
LIN {X -10.3145,Y -53.6833,Z 67,A -106.0533,B 24.8854,C -2.4713,E1 24.972,E2 189.8396} C_DIS
LIN {X -7.1477,Y -54.196,Z 67,A -102.6592,B 24.8854,C -2.4711,E1 24.9814,E2 186.4432} C_DIS
LIN {X -4.4515,Y -54.4837,Z 67,A -98.7542,B 24.8835,C -2.4915,E1 24.9924,E2 182.4878} C_DIS
LIN {X -0.9847,Y -54.6563,Z 67,A -96.4311,B 24.8858,C -2.4664,E1 24.9987,E2 180.224} C_DIS
LIN {X 0.293,Y -54.6599,Z 67,A -94.8409,B 24.8853,C -2.4717,E1 25.0032,E2 178.6214} C_DIS
Enddeposition()
LIN {X 0.293,Y -54.6599,Z 67,A -94.8409,B 24.8853,C -2.4717,E1 25.0032,E2 178.6214} C_DIS
Startdeposition()
$VEL.CP = VEL_PRINT
LIN {X -0.3288,Y -53.6767,Z 67,A -96.6339,B 24.8858,C -2.467,E1 24.9981,E2 180.4255} C_DIS
LIN {X -2.0978,Y -53.6371,Z 67,A -99.4692,B 24.8874,C -2.4493,E1 24.9901,E2 183.3033} C_DIS
LIN {X -4.9711,Y -53.447,Z 67,A -102.3312,B 24.887,C -2.4533,E1 24.9822,E2 186.1572} C_DIS
LIN {X -9.3391,Y -52.8593,Z 67,A -106.7682,B 24.8865,C -2.4593,E1 24.9699,E2 190.5838} C_DIS
LIN {X -13.6544,Y -51.9128,Z 67,A -111.0069,B 24.8855,C -2.4702,E1 24.9585,E2 194.8023} C_DIS
LIN {X -16.917,Y -50.9424,Z 67,A -115.5048,B 24.8866,C -2.4576,E1 24.9464,E2 199.3379} C_DIS
LIN {X -20.0736,Y -49.7826,Z 67,A -118.3652,B 24.8852,C -2.4736,E1 24.939,E2 202.1665} C_DIS
LIN {X -21.9813,Y -48.9706,Z 67,A -120.834,B 24.8854,C -2.4715,E1 24.9327,E2 204.6461} C_DIS
LIN {X -24.1395,Y -47.9446,Z 67,A -123.5175,B 24.8853,C -2.4722,E1 24.9259,E2 207.3349} C_DIS
LIN {X -27.4783,Y -46.1116,Z 67,A -127.2814,B 24.8843,C -2.4829,E1 24.9168,E2 211.0844} C_DIS
LIN {X -29.9159,Y -44.5688,Z 67,A -130.476,B 24.884,C -2.4856,E1 24.9093,E2 214.2827} C_DIS
LIN {X -31.6921,Y -43.3233,Z 67,A -132.5392,B 24.8833,C -2.4937,E1 24.9047,E2 216.334} C_DIS
LIN {X -33.8899,Y -41.6267,Z 67,A -136.4054,B 24.8842,C -2.4841,E1 24.8961,E2 220.2373} C_DIS
LIN {X -37.6099,Y -38.2986,Z 67,A -140.9748,B 24.882,C -2.507,E1 24.8869,E2 224.7708} C_DIS
LIN {X -39.1891,Y -36.6815,Z 67,A -143.4871,B 24.8817,C -2.5105,E1 24.882,E2 227.2856} C_DIS
LIN {X -40.7951,Y -34.8862,Z 67,A -146.4903,B 24.8818,C -2.5093,E1 24.8765,E2 230.3052} C_DIS
LIN {X -43.7578,Y -31.0896,Z 67,A -150.8251,B 24.8794,C -2.5343,E1 24.8692,E2 234.601} C_DIS
LIN {X -45.1887,Y -28.9702,Z 67,A -154.0575,B 24.8795,C -2.5332,E1 24.8642,E2 237.8523} C_DIS
LIN {X -47.2458,Y -25.4784,Z 67,A -158.0348,B 24.8779,C -2.5499,E1 24.8587,E2 241.8102} C_DIS
LIN {X -48.3791,Y -23.2542,Z 67,A -161.1169,B 24.8779,C -2.5507,E1 24.8548,E2 244.907} C_DIS
LIN {X -49.4799,Y -20.8094,Z 67,A -164.0251,B 24.8772,C -2.558,E1 24.8516,E2 247.8138} C_DIS
LIN {X -50.7321,Y -17.5388,Z 67,A -167.7275,B 24.8761,C -2.5693,E1 24.848,E2 251.5102} C_DIS
LIN {X -51.7368,Y -14.301,Z 67,A -171.4596,B 24.8752,C -2.5783,E1 24.845,E2 255.2424} C_DIS
LIN {X -52.4823,Y -11.2664,Z 67,A -174.4086,B 24.8736,C -2.5942,E1 24.8432,E2 258.1706} C_DIS
LIN {X -52.7957,Y -9.6911,Z 67,A -176.2787,B 24.8734,C -2.5971,E1 24.8422,E2 260.0449} C_DIS
LIN {X -53.1135,Y -7.7648,Z 67,A -178.4089,B 24.8728,C -2.6028,E1 24.8413,E2 262.1742} C_DIS
LIN {X -53.3669,Y -5.7637,Z 67,A 179.3422,B 24.8723,C -2.608,E1 24.8405,E2 264.424} C_DIS
LIN {X -53.5779,Y -3.2851,Z 67,A 176.568,B 24.8717,C -2.6145,E1 24.84,E2 267.1994} C_DIS
LIN {X -53.6766,Y -0.4567,Z 67,A 173.4294,B 24.8709,C -2.6222,E1 24.8398,E2 270.3383} C_DIS
LIN {X -53.6335,Y 2.1696,Z 67,A 170.5474,B 24.8701,C -2.6299,E1 24.84,E2 273.2194} C_DIS
LIN {X -53.4108,Y 5.3517,Z 67,A 167.1245,B 24.8691,C -2.6403,E1 24.8408,E2 276.6378} C_DIS
LIN {X -52.9329,Y 8.9109,Z 67,A 163.8109,B 24.8671,C -2.6602,E1 24.8422,E2 279.9238} C_DIS
LIN {X -52.5982,Y 10.7107,Z 67,A 161.0457,B 24.8677,C -2.6541,E1 24.8437,E2 282.7198} C_DIS
LIN {X -51.897,Y 13.7142,Z 67,A 158.3342,B 24.8658,C -2.673,E1 24.8455,E2 285.4019} C_DIS
LIN {X -50.9601,Y 16.8658,Z 67,A 154.1495,B 24.8658,C -2.6737,E1 24.849,E2 289.6091} C_DIS
LIN {X -49.81,Y 20.0081,Z 67,A 150.8861,B 24.8642,C -2.689,E1 24.8523,E2 292.8542} C_DIS
LIN {X -48.6028,Y 22.7825,Z 67,A 147.9969,B 24.8627,C -2.7037,E1 24.8555,E2 295.7241} C_DIS
LIN {X -47.7039,Y 24.6104,Z 67,A 145.9171,B 24.8619,C -2.7114,E1 24.8581,E2 297.7965} C_DIS
LIN {X -46.48,Y 26.8499,Z 67,A 142.356,B 24.8624,C -2.7064,E1 24.8631,E2 301.3883} C_DIS
LIN {X -44.9495,Y 29.341,Z 67,A 139.3797,B 24.8613,C -2.7172,E1 24.8675,E2 304.3539} C_DIS
LIN {X -42.6678,Y 32.5701,Z 67,A 135.5534,B 24.8596,C -2.7345,E1 24.8738,E2 308.1575} C_DIS
LIN {X -41.0563,Y 34.5799,Z 67,A 132.2212,B 24.8598,C -2.7325,E1 24.8798,E2 311.5098} C_DIS
LIN {X -39.0346,Y 36.8457,Z 67,A 129.7375,B 24.8577,C -2.7523,E1 24.8844,E2 313.9573} C_DIS
LIN {X -37.3209,Y 38.5805,Z 67,A 126.5774,B 24.858,C -2.7496,E1 24.8907,E2 317.137} C_DIS
LIN {X -35.6492,Y 40.1307,Z 67,A 124.3675,B 24.8571,C -2.7586,E1 24.8952,E2 319.3343} C_DIS
LIN {X -33.5414,Y 41.9091,Z 67,A 120.9112,B 24.8573,C -2.7568,E1 24.9028,E2 322.808} C_DIS
LIN {X -30.6564,Y 44.0622,Z 67,A 117.082,B 24.8564,C -2.7647,E1 24.9114,E2 326.6316} C_DIS
LIN {X -26.4073,Y 46.7335,Z 67,A 111.3519,B 24.8561,C -2.7682,E1 24.9252,E2 332.3707} C_DIS
LIN {X -21.7872,Y 49.058,Z 67,A 106.7706,B 24.8536,C -2.7921,E1 24.9366,E2 336.9068} C_DIS
LIN {X -19.9547,Y 49.831,Z 67,A 104.2612,B 24.8539,C -2.7886,E1 24.9431,E2 339.4302} C_DIS
LIN {X -16.6994,Y 51.0143,Z 67,A 100.6767,B 24.8533,C -2.7949,E1 24.9526,E2 343.0064} C_DIS
LIN {X -13.7228,Y 51.8942,Z 67,A 97.5351,B 24.8526,C -2.8013,E1 24.961,E2 346.1379} C_DIS
LIN {X -11.293,Y 52.4765,Z 67,A 94.7785,B 24.8526,C -2.8021,E1 24.9685,E2 348.896} C_DIS
LIN {X -8.3469,Y 53.0249,Z 67,A 91.4453,B 24.8526,C -2.8021,E1 24.9777,E2 352.2325} C_DIS
LIN {X -5.8647,Y 53.357,Z 67,A 89.0654,B 24.8518,C -2.8088,E1 24.9842,E2 354.5983} C_DIS
LIN {X -3.6346,Y 53.5545,Z 67,A 86.594,B 24.8518,C -2.8084,E1 24.9911,E2 357.0716} C_DIS
LIN {X -0.7469,Y 53.6728,Z 67,A 83.1136,B 24.8525,C -2.8022,E1 25.0009,E2 360.5671} C_DIS
LIN {X 1.9531,Y 53.643,Z 67,A 80.8937,B 24.8512,C -2.8145,E1 25.007,E2 362.7575} C_DIS
LIN {X 4.7069,Y 53.4708,Z 67,A 77.3929,B 24.8523,C -2.8043,E1 25.0168,E2 366.2809} C_DIS
LIN {X 8.2661,Y 53.0374,Z 67,A 73.3586,B 24.8528,C -2.7996,E1 25.028,E2 370.3228} C_DIS
LIN {X 11.5658,Y 52.4163,Z 67,A 69.5857,B 24.8533,C -2.7945,E1 25.0383,E2 374.1031} C_DIS
LIN {X 16.2545,Y 51.1583,Z 67,A 65.1595,B 24.8522,C -2.8051,E1 25.0501,E2 378.4966} C_DIS
LIN {X 18.3491,Y 50.4441,Z 67,A 63.0358,B 24.8519,C -2.8077,E1 25.0557,E2 380.61} C_DIS
LIN {X 20.3012,Y 49.6906,Z 67,A 60.6877,B 24.8524,C -2.8033,E1 25.0618,E2 382.9632} C_DIS
LIN {X 22.6153,Y 48.681,Z 67,A 57.5027,B 24.8537,C -2.7908,E1 25.07,E2 386.1698} C_DIS
LIN {X 24.8774,Y 47.5651,Z 67,A 55.0318,B 24.8536,C -2.7917,E1 25.0761,E2 388.6318} C_DIS
LIN {X 27.3497,Y 46.1876,Z 67,A 51.9721,B 24.8541,C -2.7868,E1 25.0835,E2 391.6941} C_DIS
LIN {X 29.4752,Y 44.8611,Z 67,A 49.4638,B 24.8542,C -2.7859,E1 25.0894,E2 394.1962} C_DIS
LIN {X 31.6774,Y 43.334,Z 67,A 46.3019,B 24.8553,C -2.7752,E1 25.0966,E2 397.3726} C_DIS
LIN {X 33.8406,Y 41.6666,Z 67,A 43.8982,B 24.8548,C -2.7802,E1 25.1018,E2 399.7554} C_DIS
LIN {X 35.4046,Y 40.3463,Z 67,A 41.5032,B 24.8557,C -2.7718,E1 25.1069,E2 402.1609} C_DIS
LIN {X 37.169,Y 38.7269,Z 67,A 38.9517,B 24.8562,C -2.7668,E1 25.1121,E2 404.7139} C_DIS
LIN {X 38.9269,Y 36.9603,Z 67,A 36.346,B 24.8567,C -2.7623,E1 25.1172,E2 407.3192} C_DIS
LIN {X 40.3343,Y 35.4184,Z 67,A 34.2187,B 24.857,C -2.7594,E1 25.1211,E2 409.4437} C_DIS
LIN {X 41.5365,Y 34.0012,Z 67,A 32.2938,B 24.8573,C -2.7561,E1 25.1246,E2 411.3678} C_DIS
LIN {X 42.9996,Y 32.1301,Z 67,A 29.2851,B 24.859,C -2.7403,E1 25.1297,E2 414.3995} C_DIS
LIN {X 44.727,Y 29.6781,Z 67,A 25.6455,B 24.8607,C -2.7233,E1 25.1354,E2 418.0614} C_DIS
LIN {X 47.0291,Y 25.8779,Z 67,A 21.2325,B 24.8613,C -2.7176,E1 25.1416,E2 422.4649} C_DIS
LIN {X 48.6479,Y 22.6865,Z 67,A 17.4456,B 24.8623,C -2.7078,E1 25.1462,E2 426.2546} C_DIS
LIN {X 49.728,Y 20.2095,Z 67,A 14.5567,B 24.8631,C -2.6996,E1 25.1492,E2 429.1471} C_DIS
LIN {X 50.9536,Y 16.8851,Z 67,A 11.0008,B 24.8638,C -2.6933,E1 25.1525,E2 432.6978} C_DIS
LIN {X 51.9829,Y 13.382,Z 67,A 7.6636,B 24.8638,C -2.6937,E1 25.155,E2 436.015} C_DIS
LIN {X 52.7059,Y 10.1672,Z 67,A 3.5412,B 24.8661,C -2.6701,E1 25.1574,E2 440.1693} C_DIS
LIN {X 53.2817,Y 6.4995,Z 67,A -0.5103,B 24.8675,C -2.656,E1 25.159,E2 444.2303} C_DIS
LIN {X 53.5702,Y 3.4031,Z 67,A -3.8531,B 24.8686,C -2.6451,E1 25.1596,E2 447.579} C_DIS
LIN {X 53.6739,Y -0.6978,Z 67,A -7.3367,B 24.8681,C -2.6505,E1 25.1598,E2 451.0289} C_DIS
LIN {X 53.4993,Y -4.3731,Z 67,A -11.2658,B 24.8693,C -2.6381,E1 25.1592,E2 454.9641} C_DIS
LIN {X 53.3391,Y -6.0202,Z 67,A -13.8216,B 24.8716,C -2.6155,E1 25.1584,E2 457.5581} C_DIS
LIN {X 52.6539,Y -10.4361,Z 67,A -17.8296,B 24.8714,C -2.6169,E1 25.1565,E2 461.5394} C_DIS
LIN {X 51.9265,Y -13.6015,Z 67,A -22.0838,B 24.8741,C -2.5892,E1 25.1537,E2 465.8344} C_DIS
LIN {X 50.827,Y -17.2605,Z 67,A -26.0636,B 24.8751,C -2.5788,E1 25.1503,E2 469.8162} C_DIS
LIN {X 49.5507,Y -20.6415,Z 67,A -29.1059,B 24.8746,C -2.5847,E1 25.1472,E2 472.8279} C_DIS
LIN {X 48.591,Y -22.8087,Z 67,A -32.2608,B 24.8766,C -2.5638,E1 25.1435,E2 476.015} C_DIS
LIN {X 47.4852,Y -25.0289,Z 67,A -34.6156,B 24.8767,C -2.5624,E1 25.1405,E2 478.3607} C_DIS
LIN {X 45.8511,Y -27.9101,Z 67,A -37.7091,B 24.8767,C -2.5618,E1 25.1362,E2 481.4397} C_DIS
LIN {X 44.8598,Y -29.4771,Z 67,A -39.9057,B 24.8778,C -2.5516,E1 25.1328,E2 483.6492} C_DIS
LIN {X 43.6076,Y -31.3001,Z 67,A -42.2895,B 24.8784,C -2.5448,E1 25.129,E2 486.0377} C_DIS
LIN {X 42.0812,Y -33.3237,Z 67,A -45.1532,B 24.8794,C -2.5343,E1 25.1241,E2 488.9125} C_DIS
LIN {X 40.5952,Y -35.1194,Z 67,A -47.3933,B 24.8795,C -2.5332,E1 25.1201,E2 491.1451} C_DIS
LIN {X 39.4469,Y -36.4042,Z 67,A -49.0827,B 24.8797,C -2.5317,E1 25.1169,E2 492.8304} C_DIS
LIN {X 37.7194,Y -38.1908,Z 67,A -52.2467,B 24.8813,C -2.5147,E1 25.1106,E2 496.0212} C_DIS
LIN {X 35.9093,Y -39.8978,Z 67,A -54.4153,B 24.8809,C -2.5187,E1 25.1062,E2 498.1716} C_DIS
LIN {X 34.6079,Y -41.0322,Z 67,A -56.2784,B 24.8813,C -2.5142,E1 25.1023,E2 500.0381} C_DIS
LIN {X 32.7868,Y -42.5008,Z 67,A -59.0546,B 24.8824,C -2.5031,E1 25.0961,E2 502.8302} C_DIS
LIN {X 30.7376,Y -44.0058,Z 67,A -61.5635,B 24.8825,C -2.5018,E1 25.0905,E2 505.3333} C_DIS
LIN {X 28.8881,Y -45.2415,Z 67,A -64.0411,B 24.8831,C -2.4952,E1 25.0847,E2 507.8185} C_DIS
LIN {X 27.3043,Y -46.2144,Z 67,A -66.2932,B 24.884,C -2.4862,E1 25.0792,E2 510.085} C_DIS
LIN {X 23.9282,Y -48.0494,Z 67,A -70.1343,B 24.8841,C -2.4846,E1 25.0697,E2 513.9191} C_DIS
LIN {X 20.0297,Y -49.8012,Z 67,A -74.3398,B 24.8841,C -2.485,E1 25.059,E2 518.1136} C_DIS
LIN {X 18.6685,Y -50.3273,Z 67,A -76.1383,B 24.8847,C -2.4781,E1 25.0543,E2 519.9244} C_DIS
LIN {X 16.5123,Y -51.0748,Z 67,A -78.3695,B 24.8847,C -2.4792,E1 25.0484,E2 522.1487} C_DIS
LIN {X 15.048,Y -51.5253,Z 67,A -80.8096,B 24.8863,C -2.4617,E1 25.0418,E2 524.6261} C_DIS
LIN {X 10.389,Y -52.6632,Z 67,A -85.2034,B 24.8854,C -2.471,E1 25.0299,E2 528.992} C_DIS
LIN {X 7.3688,Y -53.1698,Z 67,A -89.0394,B 24.8866,C -2.4578,E1 25.0192,E2 532.8555} C_DIS
LIN {X 4.0368,Y -53.5262,Z 67,A -92.0023,B 24.8857,C -2.4676,E1 25.011,E2 535.7935} C_DIS
LIN {X 1.3822,Y -53.6603,Z 67,A -95.2767,B 24.8866,C -2.4584,E1 25.0018,E2 539.0888} C_DIS
LIN {X 1.3822,Y -53.6603,Z 67,A -95.2767,B 24.8866,C -2.4584,E1 25.0018,E2 539.0888} C_DIS
Enddeposition()
LIN {X 0.2815,Y -52.6861,Z 67,A -95.777,B 24.8838,C -2.4879,E1 25.0006,E2 539.5188} C_DIS
Startdeposition()
$VEL.CP = VEL_PRINT
LIN {X 2.1617,Y -52.6459,Z 67,A -93.1189,B 24.8827,C -2.4999,E1 25.0081,E2 536.8328} C_DIS
LIN {X 3.8226,Y -52.552,Z 67,A -91.0535,B 24.8822,C -2.5055,E1 25.0139,E2 534.755} C_DIS
LIN {X 6.4309,Y -52.2966,Z 67,A -88.3019,B 24.8822,C -2.5053,E1 25.0216,E2 532.0058} C_DIS
LIN {X 8.7268,Y -51.9625,Z 67,A -85.9125,B 24.8822,C -2.5045,E1 25.0281,E2 529.6205} C_DIS
LIN {X 10.5866,Y -51.6157,Z 67,A -83.3116,B 24.8811,C -2.5168,E1 25.0353,E2 526.9936} C_DIS
LIN {X 14.3181,Y -50.7075,Z 67,A -79.5156,B 24.8814,C -2.5136,E1 25.0456,E2 523.2112} C_DIS
LIN {X 16.7314,Y -49.9633,Z 67,A -76.6673,B 24.8809,C -2.5189,E1 25.0531,E2 520.3557} C_DIS
LIN {X 19.5615,Y -48.9255,Z 67,A -73.5808,B 24.8809,C -2.5194,E1 25.0612,E2 517.2745} C_DIS
LIN {X 23.1282,Y -47.3438,Z 67,A -69.4871,B 24.8805,C -2.5228,E1 25.0716,E2 513.183} C_DIS
LIN {X 25.7436,Y -45.9731,Z 67,A -66.182,B 24.8798,C -2.5302,E1 25.0797,E2 509.8699} C_DIS
LIN {X 27.6056,Y -44.8803,Z 67,A -63.9006,B 24.8796,C -2.5331,E1 25.0852,E2 507.5886} C_DIS
LIN {X 29.0833,Y -43.9366,Z 67,A -61.7516,B 24.8787,C -2.5417,E1 25.0902,E2 505.4263} C_DIS
LIN {X 31.425,Y -42.2931,Z 67,A -58.8279,B 24.8785,C -2.5441,E1 25.0969,E2 502.5071} C_DIS
LIN {X 33.2332,Y -40.8879,Z 67,A -55.5642,B 24.8764,C -2.5655,E1 25.104,E2 499.2051} C_DIS
LIN {X 37.0219,Y -37.4918,Z 67,A -50.0533,B 24.8752,C -2.5779,E1 25.1152,E2 493.6875} C_DIS
LIN {X 40.4511,Y -33.7636,Z 67,A -45.3523,B 24.8756,C -2.5746,E1 25.1239,E2 489.0152} C_DIS
LIN {X 41.8743,Y -31.981,Z 67,A -42.7679,B 24.8747,C -2.5834,E1 25.1284,E2 486.4224} C_DIS
LIN {X 43.5424,Y -29.6705,Z 67,A -39.9203,B 24.8744,C -2.5864,E1 25.1329,E2 483.5815} C_DIS
LIN {X 44.5006,Y -28.2138,Z 67,A -37.3696,B 24.8725,C -2.6056,E1 25.1368,E2 480.9983} C_DIS
LIN {X 46.2865,Y -25.1758,Z 67,A -34.2345,B 24.8729,C -2.6016,E1 25.1411,E2 477.8888} C_DIS
LIN {X 47.538,Y -22.7247,Z 67,A -30.7994,B 24.8711,C -2.6198,E1 25.1454,E2 474.429} C_DIS
LIN {X 48.6238,Y -20.2983,Z 67,A -28.0163,B 24.8705,C -2.6261,E1 25.1484,E2 471.6463} C_DIS
LIN {X 49.7079,Y -17.4752,Z 67,A -24.9357,B 24.87,C -2.6316,E1 25.1514,E2 468.5699} C_DIS
LIN {X 50.4638,Y -15.1548,Z 67,A -21.966,B 24.8685,C -2.6466,E1 25.1539,E2 465.5816} C_DIS
LIN {X 51.4418,Y -11.4028,Z 67,A -18.2923,B 24.8683,C -2.648,E1 25.1563,E2 461.9259} C_DIS
LIN {X 51.7926,Y -9.688,Z 67,A -16.184,B 24.8673,C -2.6584,E1 25.1574,E2 459.8053} C_DIS
LIN {X 52.204,Y -7.14,Z 67,A -13.5,B 24.8667,C -2.6646,E1 25.1585,E2 457.1225} C_DIS
LIN {X 52.4718,Y -4.7927,Z 67,A -11.1565,B 24.8664,C -2.6678,E1 25.1592,E2 454.7852} C_DIS
LIN {X 52.5831,Y -3.349,Z 67,A -9.2095,B 24.865,C -2.6808,E1 25.1596,E2 452.819} C_DIS
LIN {X 52.6887,Y -0.4997,Z 67,A -5.9367,B 24.8637,C -2.6943,E1 25.1598,E2 449.5338} C_DIS
LIN {X 52.5692,Y 3.5693,Z 67,A -2.0352,B 24.8634,C -2.6969,E1 25.1593,E2 445.6495} C_DIS
LIN {X 52.3267,Y 6.1786,Z 67,A 1.3756,B 24.8613,C -2.7178,E1 25.1583,E2 442.2093} C_DIS
LIN {X 51.7063,Y 10.1364,Z 67,A 5.8393,B 24.8597,C -2.7335,E1 25.1561,E2 437.7347} C_DIS
LIN {X 50.9167,Y 13.5566,Z 67,A 9.1849,B 24.8595,C -2.7348,E1 25.1539,E2 434.4053} C_DIS
LIN {X 50.1673,Y 16.1094,Z 67,A 11.8152,B 24.8592,C -2.7377,E1 25.1517,E2 431.783} C_DIS
LIN {X 49.5375,Y 17.9528,Z 67,A 14.4336,B 24.8575,C -2.7545,E1 25.1492,E2 429.1396} C_DIS
LIN {X 48.1759,Y 21.3374,Z 67,A 17.9499,B 24.8573,C -2.7561,E1 25.1455,E2 425.6388} C_DIS
LIN {X 46.8481,Y 24.1152,Z 67,A 21.9795,B 24.8549,C -2.7797,E1 25.1404,E2 421.575} C_DIS
LIN {X 44.9922,Y 27.4219,Z 67,A 26.2286,B 24.8535,C -2.793,E1 25.1343,E2 417.316} C_DIS
LIN {X 43.1055,Y 30.3027,Z 67,A 29.3644,B 24.8538,C -2.7895,E1 25.1294,E2 414.204} C_DIS
LIN {X 41.3442,Y 32.6637,Z 67,A 32.2766,B 24.8537,C -2.7911,E1 25.1245,E2 411.3018} C_DIS
LIN {X 39.8694,Y 34.4484,Z 67,A 34.8679,B 24.8529,C -2.7984,E1 25.1198,E2 408.7052} C_DIS
LIN {X 37.8958,Y 36.6083,Z 67,A 38.4501,B 24.8513,C -2.8134,E1 25.1129,E2 405.1029} C_DIS
LIN {X 35.034,Y 39.3561,Z 67,A 42.5111,B 24.8509,C -2.8168,E1 25.1046,E2 401.0503} C_DIS
LIN {X 32.8811,Y 41.1718,Z 67,A 45.3555,B 24.8509,C -2.8181,E1 25.0985,E2 398.2138} C_DIS
LIN {X 30.9653,Y 42.6315,Z 67,A 48.3697,B 24.8495,C -2.8305,E1 25.0916,E2 395.181} C_DIS
LIN {X 28.5598,Y 44.2788,Z 67,A 50.9054,B 24.8503,C -2.8229,E1 25.0858,E2 392.6718} C_DIS
LIN {X 26.4516,Y 45.5699,Z 67,A 54.2823,B 24.8484,C -2.8403,E1 25.0776,E2 389.2639} C_DIS
LIN {X 22.5674,Y 47.6127,Z 67,A 58.9604,B 24.848,C -2.8443,E1 25.066,E2 384.5889} C_DIS
LIN {X 19.5621,Y 48.925,Z 67,A 62.4733,B 24.8477,C -2.8469,E1 25.0569,E2 381.078} C_DIS
LIN {X 16.0542,Y 50.1852,Z 67,A 66.5021,B 24.8474,C -2.8498,E1 25.0463,E2 377.0502} C_DIS
LIN {X 12.5969,Y 51.1623,Z 67,A 69.925,B 24.8481,C -2.8431,E1 25.0371,E2 373.6487} C_DIS
LIN {X 10.6013,Y 51.6127,Z 67,A 72.2207,B 24.8479,C -2.8455,E1 25.0308,E2 371.3503} C_DIS
LIN {X 8.0455,Y 52.0723,Z 67,A 75.2016,B 24.8475,C -2.8493,E1 25.0226,E2 368.3633} C_DIS
LIN {X 5.3147,Y 52.4218,Z 67,A 78.2898,B 24.8472,C -2.8516,E1 25.014,E2 365.2721} C_DIS
LIN {X 3.0163,Y 52.6039,Z 67,A 80.4364,B 24.8479,C -2.8451,E1 25.0081,E2 363.1419} C_DIS
LIN {X 1.1598,Y 52.6778,Z 67,A 82.5268,B 24.8479,C -2.8461,E1 25.0022,E2 361.0494} C_DIS
LIN {X -1.0015,Y 52.6807,Z 67,A 85.0025,B 24.8476,C -2.8478,E1 24.9953,E2 358.5695} C_DIS
LIN {X -3.0666,Y 52.6011,Z 67,A 87.056,B 24.8481,C -2.8436,E1 24.9896,E2 356.5256} C_DIS
LIN {X -5.2938,Y 52.4239,Z 67,A 89.696,B 24.8478,C -2.8462,E1 24.9822,E2 353.8782} C_DIS
LIN {X -8.349,Y 52.0243,Z 67,A 93.5194,B 24.8472,C -2.8523,E1 24.9716,E2 350.037} C_DIS
LIN {X -11.285,Y 51.4675,Z 67,A 96.4108,B 24.8481,C -2.8434,E1 24.9638,E2 347.1635} C_DIS
LIN {X -13.9261,Y 50.8167,Z 67,A 99.2061,B 24.8487,C -2.8377,E1 24.9562,E2 344.3776} C_DIS
LIN {X -15.9805,Y 50.2088,Z 67,A 102.0972,B 24.848,C -2.8447,E1 24.9485,E2 341.4648} C_DIS
LIN {X -20.1832,Y 48.6719,Z 67,A 106.3848,B 24.8497,C -2.8285,E1 24.9374,E2 337.2066} C_DIS
LIN {X -22.5158,Y 47.6376,Z 67,A 109.41,B 24.8497,C -2.8285,E1 24.9297,E2 334.1738} C_DIS
LIN {X -24.7391,Y 46.5218,Z 67,A 111.9856,B 24.8504,C -2.822,E1 24.9233,E2 331.6068} C_DIS
LIN {X -26.6638,Y 45.4455,Z 67,A 114.5647,B 24.8505,C -2.8208,E1 24.9171,E2 329.0229} C_DIS
LIN {X -29.3187,Y 43.7801,Z 67,A 117.7943,B 24.8515,C -2.8116,E1 24.9095,E2 325.8049} C_DIS
LIN {X -31.9484,Y 41.9002,Z 67,A 121.914,B 24.8512,C -2.8142,E1 24.9002,E2 321.6643} C_DIS
LIN {X -34.7391,Y 39.6164,Z 67,A 125.8033,B 24.8522,C -2.8051,E1 24.892,E2 317.7816} C_DIS
LIN {X -37.8967,Y 36.6074,Z 67,A 129.8186,B 24.8546,C -2.7825,E1 24.8841,E2 313.8036} C_DIS
LIN {X -39.6657,Y 34.6828,Z 67,A 133.46,B 24.854,C -2.7879,E1 24.8773,E2 310.1329} C_DIS
LIN {X -41.5682,Y 32.3793,Z 67,A 137.1586,B 24.8541,C -2.7866,E1 24.8709,E2 306.42} C_DIS
LIN {X -43.8733,Y 29.1793,Z 67,A 140.3366,B 24.8572,C -2.7577,E1 24.8659,E2 303.2953} C_DIS
LIN {X -45.2541,Y 26.9883,Z 67,A 143.6002,B 24.8572,C -2.7568,E1 24.8611,E2 300.0173} C_DIS
LIN {X -46.5447,Y 24.6956,Z 67,A 146.0398,B 24.8588,C -2.7422,E1 24.8579,E2 297.5998} C_DIS
LIN {X -47.9936,Y 21.7456,Z 67,A 150.6626,B 24.8582,C -2.7477,E1 24.8524,E2 292.9385} C_DIS
LIN {X -49.2058,Y 18.8436,Z 67,A 153.9644,B 24.8594,C -2.7356,E1 24.8491,E2 289.6471} C_DIS
LIN {X -50.8334,Y 13.865,Z 67,A 158.8086,B 24.8626,C -2.7052,E1 24.8451,E2 284.8477} C_DIS
LIN {X -51.31,Y 11.9816,Z 67,A 161.206,B 24.8628,C -2.703,E1 24.8435,E2 282.4417} C_DIS
LIN {X -51.8621,Y 9.3049,Z 67,A 164.1854,B 24.8637,C -2.6938,E1 24.8419,E2 279.4666} C_DIS
LIN {X -52.2921,Y 6.4658,Z 67,A 167.2798,B 24.8648,C -2.6835,E1 24.8408,E2 276.3783} C_DIS
LIN {X -52.5864,Y 3.303,Z 67,A 171.2407,B 24.8651,C -2.6803,E1 24.8399,E2 272.4013} C_DIS
LIN {X -52.6885,Y 0.5182,Z 67,A 174.3146,B 24.866,C -2.6714,E1 24.8398,E2 269.3301} C_DIS
LIN {X -52.574,Y -3.4973,Z 67,A 178.4233,B 24.8678,C -2.6538,E1 24.8403,E2 265.2388} C_DIS
LIN {X -52.2154,Y -7.0634,Z 67,A -177.9925,B 24.8694,C -2.637,E1 24.8415,E2 261.6734} C_DIS
LIN {X -51.9421,Y -8.8489,Z 67,A -175.8843,B 24.8698,C -2.6331,E1 24.8424,E2 259.5619} C_DIS
LIN {X -51.5154,Y -11.0657,Z 67,A -172.9489,B 24.8698,C -2.6331,E1 24.8441,E2 256.6095} C_DIS
LIN {X -50.3983,Y -15.3722,Z 67,A -168.4422,B 24.8718,C -2.6135,E1 24.8475,E2 252.1232} C_DIS
LIN {X -48.8015,Y -19.866,Z 67,A -163.5461,B 24.8737,C -2.5941,E1 24.8522,E2 247.2458} C_DIS
LIN {X -47.7509,Y -22.2735,Z 67,A -159.9589,B 24.8733,C -2.5976,E1 24.8563,E2 243.6308} C_DIS
LIN {X -45.9687,Y -25.7515,Z 67,A -155.9691,B 24.8748,C -2.5821,E1 24.8616,E2 239.6567} C_DIS
LIN {X -44.6983,Y -27.8984,Z 67,A -152.7154,B 24.8747,C -2.5838,E1 24.8664,E2 236.3825} C_DIS
LIN {X -43.0462,Y -30.3867,Z 67,A -149.0666,B 24.8748,C -2.5823,E1 24.8723,E2 232.7194} C_DIS
LIN {X -41.0226,Y -33.0669,Z 67,A -146.8205,B 24.8778,C -2.5511,E1 24.8761,E2 230.5371} C_DIS
LIN {X -39.4846,Y -34.8886,Z 67,A -143.7881,B 24.8778,C -2.5524,E1 24.8816,E2 227.4879} C_DIS
LIN {X -37.5048,Y -37.0088,Z 67,A -140.5735,B 24.8783,C -2.5467,E1 24.8878,E2 224.2731} C_DIS
LIN {X -35.5914,Y -38.8524,Z 67,A -136.8219,B 24.8774,C -2.5552,E1 24.8956,E2 220.4858} C_DIS
LIN {X -31.2976,Y -42.3872,Z 67,A -131.8206,B 24.8801,C -2.527,E1 24.9065,E2 215.5334} C_DIS
LIN {X -29.1126,Y -43.9173,Z 67,A -128.6787,B 24.8801,C -2.5264,E1 24.9137,E2 212.3823} C_DIS
LIN {X -27.0995,Y -45.1882,Z 67,A -126.3517,B 24.881,C -2.5182,E1 24.9193,E2 210.0676} C_DIS
LIN {X -24.9621,Y -46.4024,Z 67,A -123.4643,B 24.881,C -2.5183,E1 24.9263,E2 207.1717} C_DIS
LIN {X -22.6792,Y -47.5598,Z 67,A -120.3817,B 24.8808,C -2.5202,E1 24.9341,E2 204.0765} C_DIS
LIN {X -20.3945,Y -48.5832,Z 67,A -117.9519,B 24.8815,C -2.5123,E1 24.9403,E2 201.6599} C_DIS
LIN {X -17.2204,Y -49.7973,Z 67,A -113.9918,B 24.8814,C -2.5138,E1 24.9507,E2 197.6884} C_DIS
LIN {X -14.623,Y -50.6204,Z 67,A -111.5023,B 24.8824,C -2.5033,E1 24.9573,E2 195.2195} C_DIS
LIN {X -12.8144,Y -51.1091,Z 67,A -109.0777,B 24.8818,C -2.5091,E1 24.9639,E2 192.7776} C_DIS
LIN {X -9.5941,Y -51.8098,Z 67,A -105.8447,B 24.8826,C -2.5013,E1 24.9727,E2 189.5594} C_DIS
LIN {X -5.9397,Y -52.3547,Z 67,A -101.59,B 24.8822,C -2.5049,E1 24.9845,E2 185.2931} C_DIS
LIN {X -4.0515,Y -52.5344,Z 67,A -99.306,B 24.8818,C -2.5089,E1 24.9909,E2 182.9984} C_DIS
LIN {X -0.5462,Y -52.6878,Z 67,A -95.8138,B 24.8824,C -2.5034,E1 25.0006,E2 179.5188} C_DIS
LIN {X -0.5462,Y -52.6878,Z 67,A -95.8138,B 24.8824,C -2.5034,E1 25.0006,E2 179.5188} C_DIS
Enddeposition()
LIN {X 0.2693,Y -51.7013,Z 67,A -95.2453,B 24.8813,C -2.5147,E1 25.0023,E2 178.9236} C_DIS
Startdeposition()
$VEL.CP = VEL_PRINT
LIN {X -3.1134,Y -51.6089,Z 67,A -99.72,B 24.8826,C -2.5011,E1 24.9897,E2 183.4312} C_DIS
LIN {X -4.9966,Y -51.4613,Z 67,A -102.7673,B 24.8841,C -2.4845,E1 24.9811,E2 186.5196} C_DIS
LIN {X -7.6953,Y -51.1272,Z 67,A -105.6708,B 24.8839,C -2.487,E1 24.9731,E2 189.4194} C_DIS
LIN {X -11.9681,Y -50.2993,Z 67,A -110.1757,B 24.8832,C -2.4946,E1 24.9609,E2 193.9118} C_DIS
LIN {X -15.0721,Y -49.4577,Z 67,A -113.7686,B 24.883,C -2.4964,E1 24.9512,E2 197.5061} C_DIS
LIN {X -17.6242,Y -48.6062,Z 67,A -116.5797,B 24.8825,C -2.5017,E1 24.9438,E2 200.31} C_DIS
LIN {X -20.0571,Y -47.6538,Z 67,A -120.5238,B 24.8839,C -2.4874,E1 24.9336,E2 204.2973} C_DIS
LIN {X -23.0168,Y -46.2969,Z 67,A -122.7971,B 24.8814,C -2.5133,E1 24.928,E2 206.5146} C_DIS
LIN {X -26.1112,Y -44.6254,Z 67,A -126.5591,B 24.8807,C -2.5207,E1 24.9188,E2 210.2699} C_DIS
LIN {X -28.1037,Y -43.398,Z 67,A -129.8852,B 24.8815,C -2.5127,E1 24.9108,E2 213.6254} C_DIS
LIN {X -30.1963,Y -41.9689,Z 67,A -133.2807,B 24.8819,C -2.5081,E1 24.9031,E2 217.0438} C_DIS
LIN {X -35.1049,Y -37.9586,Z 67,A -138.8261,B 24.8785,C -2.5443,E1 24.8914,E2 222.524} C_DIS
LIN {X -36.7487,Y -36.369,Z 67,A -142.1264,B 24.8791,C -2.5376,E1 24.8847,E2 225.8543} C_DIS
LIN {X -38.7863,Y -34.1871,Z 67,A -145.5855,B 24.8787,C -2.5425,E1 24.8782,E2 229.317} C_DIS
LIN {X -40.4253,Y -32.2337,Z 67,A -148.3651,B 24.878,C -2.5497,E1 24.8734,E2 232.0924} C_DIS
LIN {X -42.4875,Y -29.4616,Z 67,A -153.0435,B 24.8783,C -2.5464,E1 24.8658,E2 236.8015} C_DIS
LIN {X -44.6743,Y -26.0283,Z 67,A -157.162,B 24.8766,C -2.5638,E1 24.8599,E2 240.8997} C_DIS
LIN {X -46.1108,Y -23.3878,Z 67,A -160.2785,B 24.8754,C -2.5759,E1 24.8559,E2 244.0038} C_DIS
LIN {X -47.5024,Y -20.4147,Z 67,A -163.9762,B 24.8745,C -2.5851,E1 24.8517,E2 247.6998} C_DIS
LIN {X -49.0479,Y -16.3554,Z 67,A -168.0378,B 24.8721,C -2.61,E1 24.8478,E2 251.7251} C_DIS
LIN {X -49.9884,Y -13.2012,Z 67,A -172.6952,B 24.8725,C -2.6062,E1 24.8442,E2 256.4183} C_DIS
LIN {X -50.7727,Y -9.7607,Z 67,A -176.2025,B 24.8707,C -2.6238,E1 24.8422,E2 259.9042} C_DIS
LIN {X -51.3928,Y -5.6474,Z 67,A 178.971,B 24.8696,C -2.635,E1 24.8405,E2 264.7328} C_DIS
LIN {X -51.664,Y -2.0008,Z 67,A 174.8828,B 24.8684,C -2.6471,E1 24.8398,E2 268.8165} C_DIS
LIN {X -51.6806,Y 1.5124,Z 67,A 171.0292,B 24.8671,C -2.66,E1 24.84,E2 272.6628} C_DIS
LIN {X -51.4669,Y 4.9357,Z 67,A 167.5917,B 24.8654,C -2.6771,E1 24.8407,E2 276.0799} C_DIS
LIN {X -51.2227,Y 7.033,Z 67,A 165.2072,B 24.8647,C -2.6838,E1 24.8415,E2 278.4626} C_DIS
LIN {X -50.8959,Y 9.0982,Z 67,A 162.491,B 24.8646,C -2.6854,E1 24.8428,E2 281.1912} C_DIS
LIN {X -50.0049,Y 13.144,Z 67,A 157.222,B 24.8641,C -2.6901,E1 24.8463,E2 286.4798} C_DIS
LIN {X -48.3211,Y 18.3914,Z 67,A 152.1273,B 24.8607,C -2.7231,E1 24.8509,E2 291.5245} C_DIS
LIN {X -47.0588,Y 21.4158,Z 67,A 147.9717,B 24.8604,C -2.7263,E1 24.8555,E2 295.6954} C_DIS
LIN {X -45.5602,Y 24.4431,Z 67,A 144.4631,B 24.8589,C -2.7405,E1 24.86,E2 299.1889} C_DIS
LIN {X -44.2227,Y 26.7867,Z 67,A 141.6428,B 24.8578,C -2.7514,E1 24.864,E2 301.9978} C_DIS
LIN {X -42.4713,Y 29.4849,Z 67,A 137.4568,B 24.8578,C -2.752,E1 24.8705,E2 306.203} C_DIS
LIN {X -40.2946,Y 32.3969,Z 67,A 133.2526,B 24.8569,C -2.7599,E1 24.8777,E2 310.4082} C_DIS
LIN {X -37.2923,Y 35.8115,Z 67,A 128.3475,B 24.8554,C -2.7742,E1 24.887,E2 315.3007} C_DIS
LIN {X -33.7599,Y 39.1603,Z 67,A 123.7941,B 24.8528,C -2.7991,E1 24.8963,E2 319.8131} C_DIS
LIN {X -31.3313,Y 41.1275,Z 67,A 119.4523,B 24.8535,C -2.7931,E1 24.9058,E2 324.1854} C_DIS
LIN {X -28.2981,Y 43.2716,Z 67,A 115.6113,B 24.8522,C -2.8052,E1 24.9147,E2 328.0103} C_DIS
LIN {X -25.9867,Y 44.6982,Z 67,A 112.9088,B 24.8511,C -2.8153,E1 24.9211,E2 330.6969} C_DIS
LIN {X -23.0182,Y 46.2958,Z 67,A 108.2126,B 24.8521,C -2.8064,E1 24.9328,E2 335.4273} C_DIS
LIN {X -17.7826,Y 48.5485,Z 67,A 101.9649,B 24.851,C -2.816,E1 24.949,E2 341.6657} C_DIS
LIN {X -14.1303,Y 49.7344,Z 67,A 98.3135,B 24.8495,C -2.8304,E1 24.9587,E2 345.289} C_DIS
LIN {X -10.5213,Y 50.621,Z 67,A 94.4329,B 24.8487,C -2.838,E1 24.9692,E2 349.1565} C_DIS
LIN {X -7.8208,Y 51.1077,Z 67,A 91.1815,B 24.8488,C -2.8367,E1 24.9782,E2 352.4142} C_DIS
LIN {X -4.7233,Y 51.4865,Z 67,A 87.4701,B 24.8491,C -2.8343,E1 24.9885,E2 356.1336} C_DIS
LIN {X -2.0088,Y 51.6641,Z 67,A 84.8153,B 24.8483,C -2.8414,E1 24.9959,E2 358.7721} C_DIS
LIN {X 0.8629,Y 51.6956,Z 67,A 81.4727,B 24.8486,C -2.8393,E1 25.0052,E2 362.1196} C_DIS
LIN {X 3.6998,Y 51.5706,Z 67,A 78.397,B 24.8484,C -2.8405,E1 25.0138,E2 365.1911} C_DIS
LIN {X 5.9888,Y 51.3547,Z 67,A 76.1299,B 24.8479,C -2.8451,E1 25.02,E2 367.4458} C_DIS
LIN {X 8.6908,Y 50.9673,Z 67,A 73.0894,B 24.848,C -2.844,E1 25.0284,E2 370.4861} C_DIS
LIN {X 10.3953,Y 50.6469,Z 67,A 70.7435,B 24.8489,C -2.8356,E1 25.0349,E2 372.8491} C_DIS
LIN {X 13.6638,Y 49.8649,Z 67,A 67.3445,B 24.8485,C -2.8393,E1 25.0441,E2 376.2342} C_DIS
LIN {X 15.8539,Y 49.2121,Z 67,A 64.708,B 24.849,C -2.8355,E1 25.0511,E2 378.8749} C_DIS
LIN {X 19.8963,Y 47.7215,Z 67,A 60.4251,B 24.8485,C -2.8402,E1 25.0623,E2 383.1376} C_DIS
LIN {X 21.9157,Y 46.8282,Z 67,A 57.1668,B 24.8504,C -2.8223,E1 25.0706,E2 386.4301} C_DIS
LIN {X 24.9031,Y 45.3109,Z 67,A 53.7763,B 24.8502,C -2.8235,E1 25.079,E2 389.8082} C_DIS
LIN {X 27.201,Y 43.9696,Z 67,A 50.9034,B 24.8505,C -2.8207,E1 25.0858,E2 392.6789} C_DIS
LIN {X 29.0508,Y 42.7695,Z 67,A 48.3474,B 24.8512,C -2.8147,E1 25.0918,E2 395.2406} C_DIS
LIN {X 31.4121,Y 41.0668,Z 67,A 45.054,B 24.8519,C -2.8079,E1 25.0992,E2 398.5384} C_DIS
LIN {X 33.7357,Y 39.1799,Z 67,A 41.1873,B 24.8537,C -2.7911,E1 25.1075,E2 402.4299} C_DIS
LIN {X 37.7216,Y 35.359,Z 67,A 36.0937,B 24.8529,C -2.7985,E1 25.1175,E2 407.4846} C_DIS
LIN {X 38.765,Y 34.2125,Z 67,A 33.9428,B 24.8542,C -2.7861,E1 25.1215,E2 409.6552} C_DIS
LIN {X 40.6369,Y 31.966,Z 67,A 30.9325,B 24.8545,C -2.7832,E1 25.1268,E2 412.6585} C_DIS
LIN {X 42.1331,Y 29.9664,Z 67,A 28.2056,B 24.8551,C -2.7773,E1 25.1313,E2 415.3862} C_DIS
LIN {X 43.59,Y 27.8047,Z 67,A 24.9937,B 24.8566,C -2.7635,E1 25.1362,E2 418.6146} C_DIS
LIN {X 45.2944,Y 24.9334,Z 67,A 21.346,B 24.8575,C -2.7548,E1 25.1413,E2 422.264} C_DIS
LIN {X 46.7379,Y 22.1096,Z 67,A 17.9433,B 24.8582,C -2.7475,E1 25.1455,E2 425.6658} C_DIS
LIN {X 48.0217,Y 19.1616,Z 67,A 14.4022,B 24.8592,C -2.7379,E1 25.1493,E2 429.2102} C_DIS
LIN {X 49.3776,Y 15.3303,Z 67,A 10.359,B 24.8596,C -2.7342,E1 25.1529,E2 433.2392} C_DIS
LIN {X 50.1907,Y 12.4134,Z 67,A 6.8916,B 24.8609,C -2.7219,E1 25.1555,E2 436.7159} C_DIS
LIN {X 50.9577,Y 8.7486,Z 67,A 2.8235,B 24.862,C -2.711,E1 25.1577,E2 440.7861} C_DIS
LIN {X 51.2228,Y 7.0322,Z 67,A 0.7695,B 24.8629,C -2.7023,E1 25.1585,E2 442.8484} C_DIS
LIN {X 51.5283,Y 4.2451,Z 67,A -1.8597,B 24.8629,C -2.7026,E1 25.1593,E2 445.4613} C_DIS
LIN {X 51.6464,Y 2.4133,Z 67,A -4.4837,B 24.8647,C -2.684,E1 25.1597,E2 448.1139} C_DIS
LIN {X 51.7031,Y -0.2888,Z 67,A -7.2459,B 24.8652,C -2.6794,E1 25.1597,E2 450.8705} C_DIS
LIN {X 51.6513,Y -2.3073,Z 67,A -9.5492,B 24.866,C -2.671,E1 25.1595,E2 453.18} C_DIS
LIN {X 51.4993,Y -4.5846,Z 67,A -12.3669,B 24.8674,C -2.657,E1 25.1589,E2 456.014} C_DIS
LIN {X 51.0336,Y -8.2947,Z 67,A -15.894,B 24.8674,C -2.6568,E1 25.1576,E2 459.5209} C_DIS
LIN {X 50.6511,Y -10.3749,Z 67,A -18.5329,B 24.8688,C -2.6433,E1 25.1562,E2 462.1763} C_DIS
LIN {X 50.0298,Y -13.0469,Z 67,A -21.664,B 24.8699,C -2.6319,E1 25.1541,E2 465.3161} C_DIS
LIN {X 49.1518,Y -16.0401,Z 67,A -25.2526,B 24.8713,C -2.6186,E1 25.1511,E2 468.9158} C_DIS
LIN {X 48.2168,Y -18.6648,Z 67,A -27.9572,B 24.8713,C -2.6171,E1 25.1485,E2 471.6087} C_DIS
LIN {X 47.0977,Y -21.3303,Z 67,A -31.6373,B 24.8733,C -2.5978,E1 25.1443,E2 475.3144} C_DIS
LIN {X 45.6964,Y -24.1872,Z 67,A -34.437,B 24.8728,C -2.6025,E1 25.1408,E2 478.0882} C_DIS
LIN {X 44.4003,Y -26.4921,Z 67,A -37.9517,B 24.8748,C -2.5822,E1 25.1359,E2 481.6328} C_DIS
LIN {X 42.8386,Y -28.9488,Z 67,A -41.1335,B 24.8756,C -2.5742,E1 25.131,E2 484.8175} C_DIS
LIN {X 40.7801,Y -31.7833,Z 67,A -44.4586,B 24.8755,C -2.5752,E1 25.1255,E2 488.1243} C_DIS
LIN {X 39.7517,Y -33.0601,Z 67,A -46.8501,B 24.8771,C -2.5589,E1 25.1212,E2 490.5434} C_DIS
LIN {X 37.6657,Y -35.4184,Z 67,A -50.3548,B 24.8779,C -2.55,E1 25.1145,E2 494.0538} C_DIS
LIN {X 34.9088,Y -38.1386,Z 67,A -54.2765,B 24.8782,C -2.5473,E1 25.1066,E2 497.9655} C_DIS
LIN {X 32.5183,Y -40.1962,Z 67,A -57.501,B 24.8784,C -2.545,E1 25.0998,E2 501.183} C_DIS
LIN {X 31.2239,Y -41.2102,Z 67,A -59.8003,B 24.8797,C -2.5318,E1 25.0946,E2 503.5054} C_DIS
LIN {X 28.3479,Y -43.2387,Z 67,A -63.3719,B 24.8797,C -2.5306,E1 25.0864,E2 507.0676} C_DIS
LIN {X 25.8217,Y -44.793,Z 67,A -67.0704,B 24.8811,C -2.5166,E1 25.0775,E2 510.7878} C_DIS
LIN {X 23.5526,Y -46.0266,Z 67,A -69.5406,B 24.8808,C -2.5194,E1 25.0714,E2 513.2444} C_DIS
LIN {X 20.6141,Y -47.4155,Z 67,A -73.4957,B 24.882,C -2.5072,E1 25.0613,E2 517.2185} C_DIS
LIN {X 17.9159,Y -48.4998,Z 67,A -76.2525,B 24.8816,C -2.5117,E1 25.0542,E2 519.9587} C_DIS
LIN {X 15.2437,Y -49.4045,Z 67,A -79.7349,B 24.8826,C -2.5013,E1 25.0449,E2 523.4592} C_DIS
LIN {X 12.2056,Y -50.2414,Z 67,A -83.0634,B 24.8826,C -2.5008,E1 25.0359,E2 526.7838} C_DIS
LIN {X 9.5321,Y -50.8163,Z 67,A -86.3394,B 24.8833,C -2.4937,E1 25.0269,E2 530.0726} C_DIS
LIN {X 5.484,Y -51.4111,Z 67,A -90.8567,B 24.8835,C -2.4912,E1 25.0144,E2 534.5923} C_DIS
LIN {X 2.4025,Y -51.647,Z 67,A -94.0103,B 24.8832,C -2.4947,E1 25.0056,E2 537.7364} C_DIS
LIN {X 0.2693,Y -51.7013,Z 67,A -95.2447,B 24.8813,C -2.5144,E1 25.0023,E2 538.9236} C_DIS
Enddeposition()
LIN {X 0.2693,Y -51.7013,Z 67,A -95.2447,B 24.8813,C -2.5144,E1 25.0023,E2 538.9236} C_DIS
Startdeposition()
$VEL.CP = VEL_PRINT
LIN {X 1.7971,Y -50.6831,Z 67,A -93.0931,B 24.8789,C -2.5396,E1 25.0085,E2 536.7125} C_DIS
LIN {X 5.0565,Y -50.4621,Z 67,A -89.2115,B 24.8784,C -2.545,E1 25.0193,E2 532.8205} C_DIS
LIN {X 7.6348,Y -50.1374,Z 67,A -86.6695,B 24.8789,C -2.5397,E1 25.0263,E2 530.2933} C_DIS
LIN {X 9.9382,Y -49.7327,Z 67,A -84.0959,B 24.8789,C -2.5405,E1 25.0334,E2 527.7206} C_DIS
LIN {X 11.9553,Y -49.286,Z 67,A -81.8841,B 24.8789,C -2.5405,E1 25.0394,E2 525.5122} C_DIS
LIN {X 14.9679,Y -48.4561,Z 67,A -77.5949,B 24.8771,C -2.5587,E1 25.0509,E2 521.187} C_DIS
LIN {X 18.1584,Y -47.3535,Z 67,A -74.0171,B 24.8771,C -2.5591,E1 25.0603,E2 517.6157} C_DIS
LIN {X 21.581,Y -45.8947,Z 67,A -69.8193,B 24.8765,C -2.5653,E1 25.071,E2 513.4137} C_DIS
LIN {X 24.8943,Y -44.1854,Z 67,A -65.9664,B 24.8765,C -2.5653,E1 25.0805,E2 509.5715} C_DIS
LIN {X 27.612,Y -42.5403,Z 67,A -61.9128,B 24.8749,C -2.5812,E1 25.0901,E2 505.4934} C_DIS
LIN {X 31.0216,Y -40.121,Z 67,A -57.8472,B 24.8752,C -2.5778,E1 25.0992,E2 501.4503} C_DIS
LIN {X 32.6851,Y -38.7779,Z 67,A -55.205,B 24.8743,C -2.5876,E1 25.1049,E2 498.795} C_DIS
LIN {X 34.7089,Y -36.9774,Z 67,A -52.2501,B 24.8738,C -2.5925,E1 25.111,E2 495.8404} C_DIS
LIN {X 36.4896,Y -35.2214,Z 67,A -49.4169,B 24.8731,C -2.5994,E1 25.1166,E2 493.0029} C_DIS
LIN {X 38.3146,Y -33.2273,Z 67,A -46.4523,B 24.8726,C -2.6053,E1 25.1221,E2 490.0378} C_DIS
LIN {X 39.6797,Y -31.5844,Z 67,A -43.5708,B 24.871,C -2.6211,E1 25.1272,E2 487.1322} C_DIS
LIN {X 42.1347,Y -28.227,Z 67,A -39.6916,B 24.8714,C -2.6169,E1 25.1334,E2 483.2817} C_DIS
LIN {X 43.1788,Y -26.6019,Z 67,A -37.1463,B 24.8701,C -2.6305,E1 25.1372,E2 480.7173} C_DIS
LIN {X 44.5501,Y -24.2348,Z 67,A -34.3801,B 24.8699,C -2.6326,E1 25.141,E2 477.9603} C_DIS
LIN {X 45.5118,Y -22.3771,Z 67,A -31.4133,B 24.8679,C -2.6519,E1 25.1447,E2 474.9636} C_DIS
LIN {X 47.0499,Y -18.9311,Z 67,A -27.5719,B 24.8675,C -2.6559,E1 25.149,E2 471.134} C_DIS
LIN {X 48.2008,Y -15.7717,Z 67,A -23.2554,B 24.8653,C -2.6782,E1 25.1529,E2 466.7888} C_DIS
LIN {X 49.0742,Y -12.7977,Z 67,A -20.3759,B 24.8655,C -2.6761,E1 25.155,E2 463.931} C_DIS
LIN {X 49.5746,Y -10.6963,Z 67,A -17.8456,B 24.8646,C -2.6856,E1 25.1566,E2 461.393} C_DIS
LIN {X 50.0706,Y -8.0621,Z 67,A -14.4116,B 24.8627,C -2.7035,E1 25.1582,E2 457.9366} C_DIS
LIN {X 50.5266,Y -4.3765,Z 67,A -10.5243,B 24.862,C -2.7103,E1 25.1594,E2 454.0563} C_DIS
LIN {X 50.6996,Y -1.2435,Z 67,A -7.3009,B 24.8616,C -2.7148,E1 25.1598,E2 450.8415} C_DIS
LIN {X 50.6939,Y 1.4737,Z 67,A -3.9241,B 24.8599,C -2.7308,E1 25.1596,E2 447.4468} C_DIS
LIN {X 50.5274,Y 4.3707,Z 67,A -0.2893,B 24.8581,C -2.7485,E1 25.1588,E2 443.7918} C_DIS
LIN {X 50.1592,Y 7.4938,Z 67,A 2.9056,B 24.8578,C -2.752,E1 25.1576,E2 440.6075} C_DIS
LIN {X 49.5798,Y 10.6722,Z 67,A 5.921,B 24.858,C -2.75,E1 25.156,E2 437.6144} C_DIS
LIN {X 49.2232,Y 12.2126,Z 67,A 8.0785,B 24.8566,C -2.763,E1 25.1546,E2 435.4386} C_DIS
LIN {X 48.5841,Y 14.5475,Z 67,A 10.7961,B 24.8558,C -2.7708,E1 25.1525,E2 432.7182} C_DIS
LIN {X 47.5784,Y 17.5603,Z 67,A 14.1685,B 24.8552,C -2.7768,E1 25.1494,E2 429.3506} C_DIS
LIN {X 46.5236,Y 20.189,Z 67,A 17.8388,B 24.8532,C -2.7954,E1 25.1455,E2 425.6563} C_DIS
LIN {X 45.648,Y 22.098,Z 67,A 20.178,B 24.8526,C -2.8013,E1 25.1426,E2 423.3159} C_DIS
LIN {X 43.8859,Y 25.4183,Z 67,A 24.0963,B 24.8521,C -2.8059,E1 25.1374,E2 419.4072} C_DIS
LIN {X 42.0678,Y 28.3258,Z 67,A 27.7508,B 24.8515,C -2.8113,E1 25.1319,E2 415.7582} C_DIS
LIN {X 41.1598,Y 29.6298,Z 67,A 29.6838,B 24.8508,C -2.8184,E1 25.1288,E2 413.8177} C_DIS
LIN {X 39.9297,Y 31.2683,Z 67,A 32.252,B 24.8497,C -2.829,E1 25.1243,E2 411.2367} C_DIS
LIN {X 37.5454,Y 34.0947,Z 67,A 37.46,B 24.8465,C -2.8588,E1 25.1146,E2 405.9813} C_DIS
LIN {X 35.0915,Y 36.6148,Z 67,A 40.4868,B 24.8476,C -2.8482,E1 25.1086,E2 402.9923} C_DIS
LIN {X 32.4067,Y 39.0108,Z 67,A 44.5947,B 24.8467,C -2.8567,E1 25.0999,E2 398.8802} C_DIS
LIN {X 29.5393,Y 41.2247,Z 67,A 48.2723,B 24.8467,C -2.8557,E1 25.0917,E2 395.2182} C_DIS
LIN {X 27.0429,Y 42.904,Z 67,A 51.3958,B 24.8467,C -2.8558,E1 25.0845,E2 392.1049} C_DIS
LIN {X 25.187,Y 44.0188,Z 67,A 54.7446,B 24.8446,C -2.8764,E1 25.0763,E2 388.7174} C_DIS
LIN {X 22.5593,Y 45.4215,Z 67,A 58.2032,B 24.8439,C -2.8823,E1 25.0677,E2 385.2541} C_DIS
LIN {X 19.8254,Y 46.6798,Z 67,A 61.0308,B 24.8447,C -2.8752,E1 25.0605,E2 382.4501} C_DIS
LIN {X 16.0315,Y 48.1151,Z 67,A 65.5371,B 24.8444,C -2.8779,E1 25.0486,E2 377.9469} C_DIS
LIN {X 12.3868,Y 49.1793,Z 67,A 70.2882,B 24.8432,C -2.889,E1 25.0358,E2 373.1769} C_DIS
LIN {X 9.1321,Y 49.8859,Z 67,A 73.528,B 24.844,C -2.8812,E1 25.027,E2 369.9597} C_DIS
LIN {X 6.4292,Y 50.3061,Z 67,A 77.0643,B 24.8431,C -2.8898,E1 25.0172,E2 366.4058} C_DIS
LIN {X 2.6034,Y 50.6487,Z 67,A 81.3183,B 24.8432,C -2.8884,E1 25.0053,E2 362.1571} C_DIS
LIN {X -1.8392,Y 50.6827,Z 67,A 86.5309,B 24.843,C -2.8905,E1 24.9908,E2 356.9392} C_DIS
LIN {X -6.1175,Y 50.3454,Z 67,A 90.787,B 24.8444,C -2.878,E1 24.979,E2 352.7105} C_DIS
LIN {X -8.6045,Y 49.9805,Z 67,A 93.4862,B 24.8448,C -2.8738,E1 24.9716,E2 350.0192} C_DIS
LIN {X -10.3092,Y 49.6565,Z 67,A 95.9404,B 24.8441,C -2.8804,E1 24.9648,E2 347.5464} C_DIS
LIN {X -14.0628,Y 48.7271,Z 67,A 99.6336,B 24.8458,C -2.865,E1 24.9549,E2 343.8844} C_DIS
LIN {X -15.7292,Y 48.2137,Z 67,A 102.3981,B 24.8446,C -2.8757,E1 24.9475,E2 341.0894} C_DIS
LIN {X -19.6823,Y 46.7402,Z 67,A 106.6169,B 24.8463,C -2.8605,E1 24.9366,E2 336.8977} C_DIS
LIN {X -22.6452,Y 45.3786,Z 67,A 110.8365,B 24.846,C -2.8634,E1 24.9259,E2 332.6605} C_DIS
LIN {X -25.7362,Y 43.7,Z 67,A 114.6498,B 24.847,C -2.854,E1 24.9167,E2 328.8584} C_DIS
LIN {X -28.0041,Y 42.2826,Z 67,A 117.3437,B 24.8481,C -2.8433,E1 24.9104,E2 326.1813} C_DIS
LIN {X -30.1393,Y 40.7886,Z 67,A 120.6559,B 24.8481,C -2.8431,E1 24.9029,E2 322.8581} C_DIS
LIN {X -33.0652,Y 38.4549,Z 67,A 124.7005,B 24.8494,C -2.8312,E1 24.8942,E2 318.8266} C_DIS
LIN {X -35.3966,Y 36.3197,Z 67,A 128.5097,B 24.8499,C -2.8266,E1 24.8864,E2 315.0127} C_DIS
LIN {X -37.6597,Y 33.9675,Z 67,A 132.2706,B 24.8507,C -2.8187,E1 24.8793,E2 311.2542} C_DIS
LIN {X -40.0263,Y 31.1446,Z 67,A 136.8331,B 24.8512,C -2.814,E1 24.8713,E2 306.6816} C_DIS
LIN {X -42.1661,Y 28.1801,Z 67,A 140.3464,B 24.8534,C -2.7937,E1 24.8658,E2 303.1995} C_DIS
LIN {X -43.5628,Y 25.967,Z 67,A 143.7394,B 24.8536,C -2.7919,E1 24.8608,E2 299.7934} C_DIS
LIN {X -45.4335,Y 22.5351,Z 67,A 147.9073,B 24.8553,C -2.7755,E1 24.8554,E2 295.6424} C_DIS
LIN {X -46.7864,Y 19.572,Z 67,A 151.3233,B 24.8568,C -2.7608,E1 24.8516,E2 292.2427} C_DIS
LIN {X -47.5366,Y 17.6743,Z 67,A 153.963,B 24.8571,C -2.7587,E1 24.849,E2 289.5933} C_DIS
LIN {X -48.5308,Y 14.7233,Z 67,A 157.6903,B 24.8579,C -2.751,E1 24.8458,E2 285.863} C_DIS
LIN {X -49.188,Y 12.3552,Z 67,A 160.593,B 24.8586,C -2.7442,E1 24.8438,E2 282.9596} C_DIS
LIN {X -49.7992,Y 9.5954,Z 67,A 163.0368,B 24.8607,C -2.7235,E1 24.8425,E2 280.551} C_DIS
LIN {X -50.1589,Y 7.4958,Z 67,A 165.8959,B 24.8608,C -2.7224,E1 24.8412,E2 277.6774} C_DIS
LIN {X -50.4944,Y 4.7276,Z 67,A 168.8534,B 24.8621,C -2.7098,E1 24.8403,E2 274.7325} C_DIS
LIN {X -50.6525,Y 2.5268,Z 67,A 171.3311,B 24.8629,C -2.7017,E1 24.8399,E2 272.2592} C_DIS
LIN {X -50.7142,Y 0.4396,Z 67,A 173.5485,B 24.8639,C -2.6922,E1 24.8398,E2 270.051} C_DIS
LIN {X -50.703,Y -1.0925,Z 67,A 175.6602,B 24.8639,C -2.6922,E1 24.8398,E2 267.9265} C_DIS
LIN {X -50.5635,Y -3.9223,Z 67,A 178.9593,B 24.8648,C -2.6837,E1 24.8405,E2 264.6281} C_DIS
LIN {X -50.2101,Y -7.1402,Z 67,A -177.6662,B 24.8663,C -2.6683,E1 24.8416,E2 261.2702} C_DIS
LIN {X -49.8623,Y -9.2657,Z 67,A -175.3499,B 24.8672,C -2.6592,E1 24.8427,E2 258.962} C_DIS
LIN {X -49.5815,Y -10.6644,Z 67,A -173.307,B 24.8671,C -2.6605,E1 24.8439,E2 256.9039} C_DIS
LIN {X -48.863,Y -13.579,Z 67,A -170.2991,B 24.8687,C -2.6448,E1 24.846,E2 253.916} C_DIS
LIN {X -48.216,Y -15.7245,Z 67,A -167.5974,B 24.8691,C -2.6399,E1 24.8483,E2 251.2106} C_DIS
LIN {X -47.1735,Y -18.6188,Z 67,A -163.8139,B 24.8697,C -2.6344,E1 24.852,E2 247.4189} C_DIS
LIN {X -46.0955,Y -21.1469,Z 67,A -160.6476,B 24.8705,C -2.6267,E1 24.8556,E2 244.2537} C_DIS
LIN {X -44.9412,Y -23.502,Z 67,A -157.1301,B 24.8705,C -2.627,E1 24.8601,E2 240.7166} C_DIS
LIN {X -43.3569,Y -26.31,Z 67,A -153.2775,B 24.871,C -2.6208,E1 24.8657,E2 236.859} C_DIS
LIN {X -40.2356,Y -30.873,Z 67,A -147.917,B 24.8739,C -2.592,E1 24.8743,E2 231.541} C_DIS
LIN {X -38.8413,Y -32.6099,Z 67,A -145.3275,B 24.8743,C -2.5874,E1 24.8789,E2 228.9506} C_DIS
Enddeposition()
END
